{region " SIGNAL AREA : NAME->C_BMS_Wkup LENGTH->2 STARTBIT :44"}
_FB_CanTx_Message_Unpack_430.S_Bit_44		:= (GVL.IOVD.C_BMS_Wkup.x OR GVL.IOVD.C_BMS_Wkup.na) AND NOT GVL.IOVD.C_BMS_Wkup.e; 
_FB_CanTx_Message_Unpack_430.S_Bit_45		:= NOT GVL.IOVD.C_BMS_Wkup.v OR GVL.IOVD.C_BMS_Wkup.na OR GVL.IOVD.C_BMS_Wkup.e; 
{endregion}

{region " SIGNAL AREA : NAME->Z_Bat_Mode LENGTH->8 STARTBIT :48"}
_FB_CanTx_Message_Unpack_430.X_Byte_6					:=
(*SELECT 1 : Is data valid and range is not exceed?*)	SEL((GVL.IOVD.Z_Bat_Mode.v AND NOT GVL.IOVD.Z_Bat_Mode.RangeExcd),
(*SELECT 2 : Is NOT AVAILABLE ?*)						SEL(GVL.IOVD.Z_Bat_Mode.na,
(*SELECT 3 : Is ERROR active ?*)						SEL(GVL.IOVD.Z_Bat_Mode.e,
(*DEFAULT VALUE assignment*)							0,
(*ERROR is active*)										16#E),
(*NOT AVAILABLE is active*)								16#F),
(*Transmission is VALID*)								GVL.IOVD.Z_Bat_Mode.x);
{endregion}

{region " SIGNAL AREA : NAME->Z_ESS_Stat LENGTH->8 STARTBIT :56"}

_FB_CanTx_Message_Unpack_430.X_Byte_7					:=
(*SELECT 1 : Is data valid and range is not exceed?*)	SEL((GVL.IOVD.Z_ESS_Stat.v AND NOT GVL.IOVD.Z_ESS_Stat.RangeExcd),
(*SELECT 2 : Is NOT AVAILABLE ?*)						SEL(GVL.IOVD.Z_ESS_Stat.na,
(*SELECT 3 : Is ERROR active ?*)						SEL(GVL.IOVD.Z_ESS_Stat.e,
(*DEFAULT VALUE assignment*)							0,
(*ERROR is active*)										16#E),
(*NOT AVAILABLE is active*)								16#F),
(*Transmission is VALID*)								GVL.IOVD.Z_ESS_Stat.x);
{endregion}

_FB_CanTx_Message_Unpack_430.S_Bit_2 	:= TRUE;
_FB_CanTx_Message_Unpack_430.S_Bit_3 	:= TRUE;
_FB_CanTx_Message_Unpack_430.S_Bit_14 	:= TRUE;
_FB_CanTx_Message_Unpack_430.S_Bit_15 	:= TRUE;
_FB_CanTx_Message_Unpack_430.S_Bit_18	:= TRUE;
_FB_CanTx_Message_Unpack_430.S_Bit_19	:= TRUE;
_FB_CanTx_Message_Unpack_430.S_Bit_20	:= TRUE;
_FB_CanTx_Message_Unpack_430.S_Bit_21	:= TRUE;
_FB_CanTx_Message_Unpack_430.S_Bit_22	:= TRUE;
_FB_CanTx_Message_Unpack_430.S_Bit_23	:= TRUE;
_FB_CanTx_Message_Unpack_430.S_Bit_28	:= TRUE;
_FB_CanTx_Message_Unpack_430.S_Bit_29	:= TRUE;
_FB_CanTx_Message_Unpack_430.S_Bit_30	:= TRUE;
_FB_CanTx_Message_Unpack_430.S_Bit_31	:= TRUE;
_FB_CanTx_Message_Unpack_430.S_Bit_46	:= TRUE;
_FB_CanTx_Message_Unpack_430.S_Bit_47	:= TRUE;

_FB_CanTx_Message_Unpack_430 (		C_Enable		:= GVL.IOVD.C_En_ESS_Durum_0X430,
     								Obj_CAN			:= ADR(GVL.IC.Obj_CAN0),
     								X_MsgID			:= 16#430,
     								Tm_CycleTime	:= TIME#500MS,
     								N_Msg_Dlc		:= 8,
     								S_Extended		:= 0,
     								S_Sent_Ok   	=> GVL.IOVD.S_SentOk_ESS_Durum_0X430);
{endregion}
//-----------------------------------------------------------------------------------------------------------------------------
//-----------------------------------------------------------------------------------------------------------------------------
{region " MESSAGE AREA :ESS_Paket_Voltaji- ID:431"}

{region " SIGNAL AREA : NAME->X_U_Bat_1 LENGTH->16 STARTBIT :0"}
_FB_UNPACK_WORD_TO_BYTE_0 (
		X_WORD_0										:= 
(*SELECT 1 : Is data valid and range is not exceed?*)	SEL((GVL.IOVD.X_U_Bat_1.v AND NOT GVL.IOVD.X_U_Bat_1.RangeExcd),
(*SELECT 2 : Is NOT AVAILABLE ?*)						SEL(GVL.IOVD.X_U_Bat_1.na,
(*SELECT 3 : Is ERROR active ?*)						SEL(GVL.IOVD.X_U_Bat_1.e,
(*DEFAULT VALUE assignment*)							0,
(*ERROR is active*)										16#FEFE),
(*NOT AVAILABLE is active*)								16#FFFF),
(*Transmission is VALID*)								UINT_TO_WORD(REAL_TO_UINT((GVL.IOVD.X_U_Bat_1.x)/0.02))),
		X_BYTE_0										=> _FB_CanTx_Message_Unpack_431.X_Byte_0,
		X_BYTE_1										=> _FB_CanTx_Message_Unpack_431.X_Byte_1);
{endregion}

{region " SIGNAL AREA : NAME->X_U_Bat_2 LENGTH->16 STARTBIT :16"}
_FB_UNPACK_WORD_TO_BYTE_1 (
		X_WORD_0										:= 
(*SELECT 1 : Is data valid and range is not exceed?*)	SEL((GVL.IOVD.X_U_Bat_2.v AND NOT GVL.IOVD.X_U_Bat_2.RangeExcd),
(*SELECT 2 : Is NOT AVAILABLE ?*)						SEL(GVL.IOVD.X_U_Bat_2.na,
(*SELECT 3 : Is ERROR active ?*)						SEL(GVL.IOVD.X_U_Bat_2.e,
(*DEFAULT VALUE assignment*)							0,
(*ERROR is active*)										16#FEFE),
(*NOT AVAILABLE is active*)								16#FFFF),
(*Transmission is VALID*)								UINT_TO_WORD(REAL_TO_UINT((GVL.IOVD.X_U_Bat_2.x)/0.02))),
		X_BYTE_0										=> _FB_CanTx_Message_Unpack_431.X_Byte_2,
		X_BYTE_1										=> _FB_CanTx_Message_Unpack_431.X_Byte_3);
{endregion}

{region " SIGNAL AREA : NAME->X_U_Bat_3 LENGTH->16 STARTBIT :32"}
_FB_UNPACK_WORD_TO_BYTE_2 (
		X_WORD_0										:= 
(*SELECT 1 : Is data valid and range is not exceed?*)	SEL((GVL.IOVD.X_U_Bat_3.v AND NOT GVL.IOVD.X_U_Bat_3.RangeExcd),
(*SELECT 2 : Is NOT AVAILABLE ?*)						SEL(GVL.IOVD.X_U_Bat_3.na,
(*SELECT 3 : Is ERROR active ?*)						SEL(GVL.IOVD.X_U_Bat_3.e,
(*DEFAULT VALUE assignment*)							0,
(*ERROR is active*)										16#FEFE),
(*NOT AVAILABLE is active*)								16#FFFF),
(*Transmission is VALID*)								UINT_TO_WORD(REAL_TO_UINT((GVL.IOVD.X_U_Bat_3.x)/0.02))),
		X_BYTE_0										=> _FB_CanTx_Message_Unpack_431.X_Byte_4,
		X_BYTE_1										=> _FB_CanTx_Message_Unpack_431.X_Byte_5);
{endregion}

{region " SIGNAL AREA : NAME->X_U_Bat_4 LENGTH->16 STARTBIT :48"}
_FB_UNPACK_WORD_TO_BYTE_3 (
		X_WORD_0										:= 
(*SELECT 1 : Is data valid and range is not exceed?*)	SEL((GVL.IOVD.X_U_Bat_4.v AND NOT GVL.IOVD.X_U_Bat_4.RangeExcd),
(*SELECT 2 : Is NOT AVAILABLE ?*)						SEL(GVL.IOVD.X_U_Bat_4.na,
(*SELECT 3 : Is ERROR active ?*)						SEL(GVL.IOVD.X_U_Bat_4.e,
(*DEFAULT VALUE assignment*)							0,
(*ERROR is active*)										16#FEFE),
(*NOT AVAILABLE is active*)								16#FFFF),
(*Transmission is VALID*)								UINT_TO_WORD(REAL_TO_UINT((GVL.IOVD.X_U_Bat_4.x)/0.02))),
		X_BYTE_0										=> _FB_CanTx_Message_Unpack_431.X_Byte_6,
		X_BYTE_1										=> _FB_CanTx_Message_Unpack_431.X_Byte_7);
{endregion}

_FB_CanTx_Message_Unpack_431 (		C_Enable		:= GVL.IOVD.C_En_ESS_Paket_Voltaji_0X431,
     								Obj_CAN			:= ADR(GVL.IC.Obj_CAN0),
     								X_MsgID			:= 16#431,
     								Tm_CycleTime	:= TIME#500MS,
     								N_Msg_Dlc		:= 8,
     								S_Extended		:= 0,
     								S_Sent_Ok   	=> GVL.IOVD.S_SentOk_ESS_Paket_Voltaji_0X431);
{endregion}
//-----------------------------------------------------------------------------------------------------------------------------
//-----------------------------------------------------------------------------------------------------------------------------
{region " MESSAGE AREA :ESS_Paket_Akim- ID:432"}

{region " SIGNAL AREA : NAME->X_I_Bat_1 LENGTH->16 STARTBIT :0"}
_FB_UNPACK_WORD_TO_BYTE_4 (
		X_WORD_0										:= 
(*SELECT 1 : Is data valid and range is not exceed?*)	SEL((GVL.IOVD.X_I_Bat_1.v AND NOT GVL.IOVD.X_I_Bat_1.RangeExcd),
(*SELECT 2 : Is NOT AVAILABLE ?*)						SEL(GVL.IOVD.X_I_Bat_1.na,
(*SELECT 3 : Is ERROR active ?*)						SEL(GVL.IOVD.X_I_Bat_1.e,
(*DEFAULT VALUE assignment*)							UINT_TO_WORD(REAL_TO_UINT((3276.8)/0.1)),
(*ERROR is active*)										16#FEFE),
(*NOT AVAILABLE is active*)								16#FFFF),
(*Transmission is VALID*)								UINT_TO_WORD(REAL_TO_UINT((GVL.IOVD.X_I_Bat_1.x + 3276.8) / 0.1))),
		X_BYTE_0										=> _FB_CanTx_Message_432.X_Byte_0,
		X_BYTE_1										=> _FB_CanTx_Message_432.X_Byte_1);
{endregion}

{region " SIGNAL AREA : NAME->X_I_Bat_2 LENGTH->16 STARTBIT :16"}
_FB_UNPACK_WORD_TO_BYTE_5 (
		X_WORD_0										:= 
(*SELECT 1 : Is data valid and range is not exceed?*)	SEL((GVL.IOVD.X_I_Bat_2.v AND NOT GVL.IOVD.X_I_Bat_2.RangeExcd),
(*SELECT 2 : Is NOT AVAILABLE ?*)						SEL(GVL.IOVD.X_I_Bat_2.na,
(*SELECT 3 : Is ERROR active ?*)						SEL(GVL.IOVD.X_I_Bat_2.e,
(*DEFAULT VALUE assignment*)							UINT_TO_WORD(REAL_TO_UINT((3276.8)/0.1)),
(*ERROR is active*)										16#FEFE),
(*NOT AVAILABLE is active*)								16#FFFF),
(*Transmission is VALID*)								UINT_TO_WORD(REAL_TO_UINT((GVL.IOVD.X_I_Bat_2.x + 3276.8) / 0.1))),
		X_BYTE_0										=> _FB_CanTx_Message_432.X_Byte_2,
		X_BYTE_1										=> _FB_CanTx_Message_432.X_Byte_3);
{endregion}

{region " SIGNAL AREA : NAME->X_I_Bat_3 LENGTH->16 STARTBIT :32"}
_FB_UNPACK_WORD_TO_BYTE_6 (
		X_WORD_0										:= 
(*SELECT 1 : Is data valid and range is not exceed?*)	SEL((GVL.IOVD.X_I_Bat_3.v AND NOT GVL.IOVD.X_I_Bat_3.RangeExcd),
(*SELECT 2 : Is NOT AVAILABLE ?*)						SEL(GVL.IOVD.X_I_Bat_3.na,
(*SELECT 3 : Is ERROR active ?*)						SEL(GVL.IOVD.X_I_Bat_3.e,
(*DEFAULT VALUE assignment*)							UINT_TO_WORD(REAL_TO_UINT((3276.8)/0.1)),
(*ERROR is active*)										16#FEFE),
(*NOT AVAILABLE is active*)								16#FFFF),
(*Transmission is VALID*)								UINT_TO_WORD(REAL_TO_UINT((GVL.IOVD.X_I_Bat_3.x + 3276.8) / 0.1))),
		X_BYTE_0										=> _FB_CanTx_Message_432.X_Byte_4,
		X_BYTE_1										=> _FB_CanTx_Message_432.X_Byte_5);
{endregion}

{region " SIGNAL AREA : NAME->X_I_Bat_4 LENGTH->16 STARTBIT :48"}
_FB_UNPACK_WORD_TO_BYTE_7 (
		X_WORD_0										:= 
(*SELECT 1 : Is data valid and range is not exceed?*)	SEL((GVL.IOVD.X_I_Bat_4.v AND NOT GVL.IOVD.X_I_Bat_4.RangeExcd),
(*SELECT 2 : Is NOT AVAILABLE ?*)						SEL(GVL.IOVD.X_I_Bat_4.na,
(*SELECT 3 : Is ERROR active ?*)						SEL(GVL.IOVD.X_I_Bat_4.e,
(*DEFAULT VALUE assignment*)							UINT_TO_WORD(REAL_TO_UINT((3276.8)/0.1)),
(*ERROR is active*)										16#FEFE),
(*NOT AVAILABLE is active*)								16#FFFF),
(*Transmission is VALID*)								UINT_TO_WORD(REAL_TO_UINT((GVL.IOVD.X_I_Bat_4.x + 3276.8) / 0.1))),
		X_BYTE_0										=> _FB_CanTx_Message_432.X_Byte_6,
		X_BYTE_1										=> _FB_CanTx_Message_432.X_Byte_7);
{endregion}

_FB_CanTx_Message_432 (		C_Enable		:= GVL.IOVD.C_En_ESS_Paket_Akim_0X432,
     						Obj_CAN			:= ADR(GVL.IC.Obj_CAN0),
     						X_MsgID			:= 16#432,
     						Tm_CycleTime	:= TIME#500MS,
     						N_Msg_Dlc		:= 8,
     						S_Extended		:= 0,
     						S_Sent_Ok  	 	=> GVL.IOVD.S_SentOk_ESS_Paket_Akim_0X432);
{endregion}
//-----------------------------------------------------------------------------------------------------------------------------
//-----------------------------------------------------------------------------------------------------------------------------
{region " MESSAGE AREA :ESS_Maksimum_Hucre_Voltaji- ID:433"}

{region " SIGNAL AREA : NAME->X_U_Max_Cell_1 LENGTH->16 STARTBIT :0"}
_FB_UNPACK_WORD_TO_BYTE_8 (
		X_WORD_0										:= 
(*SELECT 1 : Is data valid and range is not exceed?*)	SEL((GVL.IOVD.X_U_Max_Bat_1.v AND NOT GVL.IOVD.X_U_Max_Bat_1.RangeExcd),
(*SELECT 2 : Is NOT AVAILABLE ?*)						SEL(GVL.IOVD.X_U_Max_Bat_1.na,
(*SELECT 3 : Is ERROR active ?*)						SEL(GVL.IOVD.X_U_Max_Bat_1.e,
(*DEFAULT VALUE assignment*)							0,
(*ERROR is active*)										16#FEFE),
(*NOT AVAILABLE is active*)								16#FFFF),
(*Transmission is VALID*)								UINT_TO_WORD(REAL_TO_UINT((GVL.IOVD.X_U_Max_Bat_1.x) / 0.1))),
		X_BYTE_0										=> _FB_CanTx_Message_433.X_Byte_0,
		X_BYTE_1										=> _FB_CanTx_Message_433.X_Byte_1);
{endregion}

{region " SIGNAL AREA : NAME->X_U_Max_Cell_2 LENGTH->16 STARTBIT :16"}
_FB_UNPACK_WORD_TO_BYTE_9 (
		X_WORD_0										:= 
(*SELECT 1 : Is data valid and range is not exceed?*)	SEL((GVL.IOVD.X_U_Max_Bat_2.v AND NOT GVL.IOVD.X_U_Max_Bat_2.RangeExcd),
(*SELECT 2 : Is NOT AVAILABLE ?*)						SEL(GVL.IOVD.X_U_Max_Bat_2.na,
(*SELECT 3 : Is ERROR active ?*)						SEL(GVL.IOVD.X_U_Max_Bat_2.e,
(*DEFAULT VALUE assignment*)							0,
(*ERROR is active*)										16#FEFE),
(*NOT AVAILABLE is active*)								16#FFFF),
(*Transmission is VALID*)								UINT_TO_WORD(REAL_TO_UINT((GVL.IOVD.X_U_Max_Bat_2.x) / 0.1))),
		X_BYTE_0										=> _FB_CanTx_Message_433.X_Byte_2,
		X_BYTE_1										=> _FB_CanTx_Message_433.X_Byte_3);
{endregion}

{region " SIGNAL AREA : NAME->X_U_Max_Cell_3 LENGTH->16 STARTBIT :32"}
_FB_UNPACK_WORD_TO_BYTE_10 (
		X_WORD_0										:= 
(*SELECT 1 : Is data valid and range is not exceed?*)	SEL((GVL.IOVD.X_U_Max_Bat_3.v AND NOT GVL.IOVD.X_U_Max_Bat_3.RangeExcd),
(*SELECT 2 : Is NOT AVAILABLE ?*)						SEL(GVL.IOVD.X_U_Max_Bat_3.na,
(*SELECT 3 : Is ERROR active ?*)						SEL(GVL.IOVD.X_U_Max_Bat_3.e,
(*DEFAULT VALUE assignment*)							0,
(*ERROR is active*)										16#FEFE),
(*NOT AVAILABLE is active*)								16#FFFF),
(*Transmission is VALID*)								UINT_TO_WORD(REAL_TO_UINT((GVL.IOVD.X_U_Max_Bat_3.x) / 0.1))),
		X_BYTE_0										=> _FB_CanTx_Message_433.X_Byte_4,
		X_BYTE_1										=> _FB_CanTx_Message_433.X_Byte_5);
{endregion}

{region " SIGNAL AREA : NAME->X_U_Max_Cell_4 LENGTH->16 STARTBIT :48"}
_FB_UNPACK_WORD_TO_BYTE_11 (
		X_WORD_0										:= 
(*SELECT 1 : Is data valid and range is not exceed?*)	SEL((GVL.IOVD.X_U_Max_Bat_4.v AND NOT GVL.IOVD.X_U_Max_Bat_4.RangeExcd),
(*SELECT 2 : Is NOT AVAILABLE ?*)						SEL(GVL.IOVD.X_U_Max_Bat_4.na,
(*SELECT 3 : Is ERROR active ?*)						SEL(GVL.IOVD.X_U_Max_Bat_4.e,
(*DEFAULT VALUE assignment*)							0,
(*ERROR is active*)										16#FEFE),
(*NOT AVAILABLE is active*)								16#FFFF),
(*Transmission is VALID*)								UINT_TO_WORD(REAL_TO_UINT((GVL.IOVD.X_U_Max_Bat_4.x) / 0.1))),
		X_BYTE_0										=> _FB_CanTx_Message_433.X_Byte_6,
		X_BYTE_1										=> _FB_CanTx_Message_433.X_Byte_7);
{endregion}

_FB_CanTx_Message_433 (		C_Enable		:= GVL.IOVD.C_En_ESS_Maksimum_Hucre_Voltaji_0X433,
     						Obj_CAN			:= ADR(GVL.IC.Obj_CAN0),
     						X_MsgID			:= 16#433,
     						Tm_CycleTime	:= TIME#500MS,
     						N_Msg_Dlc		:= 8,
     						S_Extended		:= 0,
     						S_Sent_Ok   	=> GVL.IOVD.S_SentOk_ESS_Maksimum_Hucre_Voltaji_0X433);
{endregion}
//-----------------------------------------------------------------------------------------------------------------------------
//-----------------------------------------------------------------------------------------------------------------------------
{region " MESSAGE AREA :ESS_Minimum_Hucre_Voltaji- ID:434"}

{region " SIGNAL AREA : NAME->X_U_Min_Cell_1 LENGTH->16 STARTBIT :0"}
_FB_UNPACK_WORD_TO_BYTE_12 (
		X_WORD_0										:= 
(*SELECT 1 : Is data valid and range is not exceed?*)	SEL((GVL.IOVD.X_U_Min_Bat_1.v AND NOT GVL.IOVD.X_U_Min_Bat_1.RangeExcd),
(*SELECT 2 : Is NOT AVAILABLE ?*)						SEL(GVL.IOVD.X_U_Min_Bat_1.na,
(*SELECT 3 : Is ERROR active ?*)						SEL(GVL.IOVD.X_U_Min_Bat_1.e,
(*DEFAULT VALUE assignment*)							0,
(*ERROR is active*)										16#FEFE),
(*NOT AVAILABLE is active*)								16#FFFF),
(*Transmission is VALID*)								UINT_TO_WORD(REAL_TO_UINT((GVL.IOVD.X_U_Min_Bat_1.x) / 0.1))),
		X_BYTE_0										=> _FB_CanTx_Message_Unpack_434.X_Byte_0,
		X_BYTE_1										=> _FB_CanTx_Message_Unpack_434.X_Byte_1);
{endregion}

{region " SIGNAL AREA : NAME->X_U_Min_Cell_2 LENGTH->16 STARTBIT :16"}
_FB_UNPACK_WORD_TO_BYTE_13 (
		X_WORD_0										:= 
(*SELECT 1 : Is data valid and range is not exceed?*)	SEL((GVL.IOVD.X_U_Min_Bat_2.v AND NOT GVL.IOVD.X_U_Min_Bat_2.RangeExcd),
(*SELECT 2 : Is NOT AVAILABLE ?*)						SEL(GVL.IOVD.X_U_Min_Bat_2.na,
(*SELECT 3 : Is ERROR active ?*)						SEL(GVL.IOVD.X_U_Min_Bat_2.e,
(*DEFAULT VALUE assignment*)							0,
(*ERROR is active*)										16#FEFE),
(*NOT AVAILABLE is active*)								16#FFFF),
(*Transmission is VALID*)								UINT_TO_WORD(REAL_TO_UINT((GVL.IOVD.X_U_Min_Bat_2.x) / 0.1))),
		X_BYTE_0										=> _FB_CanTx_Message_Unpack_434.X_Byte_2,
		X_BYTE_1										=> _FB_CanTx_Message_Unpack_434.X_Byte_3);
{endregion}

{region " SIGNAL AREA : NAME->X_U_Min_Cell_3 LENGTH->16 STARTBIT :32"}
_FB_UNPACK_WORD_TO_BYTE_14 (
		X_WORD_0										:= 
(*SELECT 1 : Is data valid and range is not exceed?*)	SEL((GVL.IOVD.X_U_Min_Bat_3.v AND NOT GVL.IOVD.X_U_Min_Bat_3.RangeExcd),
(*SELECT 2 : Is NOT AVAILABLE ?*)						SEL(GVL.IOVD.X_U_Min_Bat_3.na,
(*SELECT 3 : Is ERROR active ?*)						SEL(GVL.IOVD.X_U_Min_Bat_3.e,
(*DEFAULT VALUE assignment*)							0,
(*ERROR is active*)										16#FEFE),
(*NOT AVAILABLE is active*)								16#FFFF),
(*Transmission is VALID*)								UINT_TO_WORD(REAL_TO_UINT((GVL.IOVD.X_U_Min_Bat_3.x) / 0.1))),
		X_BYTE_0										=> _FB_CanTx_Message_Unpack_434.X_Byte_4,
		X_BYTE_1										=> _FB_CanTx_Message_Unpack_434.X_Byte_5);
{endregion}

{region " SIGNAL AREA : NAME->X_U_Min_Cell_4 LENGTH->16 STARTBIT :48"}
_FB_UNPACK_WORD_TO_BYTE_15 (
		X_WORD_0										:= 
(*SELECT 1 : Is data valid and range is not exceed?*)	SEL((GVL.IOVD.X_U_Min_Bat_4.v AND NOT GVL.IOVD.X_U_Min_Bat_4.RangeExcd),
(*SELECT 2 : Is NOT AVAILABLE ?*)						SEL(GVL.IOVD.X_U_Min_Bat_4.na,
(*SELECT 3 : Is ERROR active ?*)						SEL(GVL.IOVD.X_U_Min_Bat_4.e,
(*DEFAULT VALUE assignment*)							0,
(*ERROR is active*)										16#FEFE),
(*NOT AVAILABLE is active*)								16#FFFF),
(*Transmission is VALID*)								UINT_TO_WORD(REAL_TO_UINT((GVL.IOVD.X_U_Min_Bat_4.x) / 0.1))),
		X_BYTE_0										=> _FB_CanTx_Message_Unpack_434.X_Byte_6,
		X_BYTE_1										=> _FB_CanTx_Message_Unpack_434.X_Byte_7);
{endregion}

_FB_CanTx_Message_Unpack_434 (		C_Enable		:= GVL.IOVD.C_En_ESS_Minimum_Hucre_Voltaji_0X434,
     								Obj_CAN			:= ADR(GVL.IC.Obj_CAN0),
     								X_MsgID			:= 16#434,
     								Tm_CycleTime	:= TIME#500MS,
     								N_Msg_Dlc		:= 8,
     								S_Extended		:= 0,
     								S_Sent_Ok   	=> GVL.IOVD.S_SentOk_ESS_Minimum_Hucre_Voltaji_0X434);
{endregion}
//-----------------------------------------------------------------------------------------------------------------------------
//-----------------------------------------------------------------------------------------------------------------------------
{region " MESSAGE AREA :ESS_Ortalama_Hucre_Voltaji- ID:435"}

{region " SIGNAL AREA : NAME->X_U_Avg_Cell_1 LENGTH->16 STARTBIT :0"}
_FB_UNPACK_WORD_TO_BYTE_16 (
		X_WORD_0										:= 
(*SELECT 1 : Is data valid and range is not exceed?*)	SEL((GVL.IOVD.X_U_Avg_Cell_1.v AND NOT GVL.IOVD.X_U_Avg_Cell_1.RangeExcd),
(*SELECT 2 : Is NOT AVAILABLE ?*)						SEL(GVL.IOVD.X_U_Avg_Cell_1.na,
(*SELECT 3 : Is ERROR active ?*)						SEL(GVL.IOVD.X_U_Avg_Cell_1.e,
(*DEFAULT VALUE assignment*)							0,
(*ERROR is active*)										16#FEFE),
(*NOT AVAILABLE is active*)								16#FFFF),
(*Transmission is VALID*)								UINT_TO_WORD(REAL_TO_UINT((GVL.IOVD.X_U_Avg_Cell_1.x)/0.01))),
		X_BYTE_0										=> _FB_CanTx_Message_435.X_Byte_0,
		X_BYTE_1										=> _FB_CanTx_Message_435.X_Byte_1);
{endregion}

{region " SIGNAL AREA : NAME->X_U_Avg_Cell_2 LENGTH->16 STARTBIT :16"}
_FB_UNPACK_WORD_TO_BYTE_17 (
		X_WORD_0										:= 
(*SELECT 1 : Is data valid and range is not exceed?*)	SEL((GVL.IOVD.X_U_Avg_Cell_2.v AND NOT GVL.IOVD.X_U_Avg_Cell_2.RangeExcd),
(*SELECT 2 : Is NOT AVAILABLE ?*)						SEL(GVL.IOVD.X_U_Avg_Cell_2.na,
(*SELECT 3 : Is ERROR active ?*)						SEL(GVL.IOVD.X_U_Avg_Cell_2.e,
(*DEFAULT VALUE assignment*)							0,
(*ERROR is active*)										16#FEFE),
(*NOT AVAILABLE is active*)								16#FFFF),
(*Transmission is VALID*)								UINT_TO_WORD(REAL_TO_UINT((GVL.IOVD.X_U_Avg_Cell_2.x)/0.01))),
		X_BYTE_0										=> _FB_CanTx_Message_435.X_Byte_2,
		X_BYTE_1										=> _FB_CanTx_Message_435.X_Byte_3);
{endregion}

{region " SIGNAL AREA : NAME->X_U_Avg_Cell_3 LENGTH->16 STARTBIT :32"}
_FB_UNPACK_WORD_TO_BYTE_18 (
		X_WORD_0										:= 
(*SELECT 1 : Is data valid and range is not exceed?*)	SEL((GVL.IOVD.X_U_Avg_Cell_3.v AND NOT GVL.IOVD.X_U_Avg_Cell_3.RangeExcd),
(*SELECT 2 : Is NOT AVAILABLE ?*)						SEL(GVL.IOVD.X_U_Avg_Cell_3.na,
(*SELECT 3 : Is ERROR active ?*)						SEL(GVL.IOVD.X_U_Avg_Cell_3.e,
(*DEFAULT VALUE assignment*)							0,
(*ERROR is active*)										16#FEFE),
(*NOT AVAILABLE is active*)								16#FFFF),
(*Transmission is VALID*)								UINT_TO_WORD(REAL_TO_UINT((GVL.IOVD.X_U_Avg_Cell_3.x)/0.01))),
		X_BYTE_0										=> _FB_CanTx_Message_435.X_Byte_4,
		X_BYTE_1										=> _FB_CanTx_Message_435.X_Byte_5);
{endregion}

{region " SIGNAL AREA : NAME->X_U_Avg_Cell_4 LENGTH->16 STARTBIT :48"}
_FB_UNPACK_WORD_TO_BYTE_19 (
		X_WORD_0										:= 
(*SELECT 1 : Is data valid and range is not exceed?*)	SEL((GVL.IOVD.X_U_Avg_Cell_4.v AND NOT GVL.IOVD.X_U_Avg_Cell_4.RangeExcd),
(*SELECT 2 : Is NOT AVAILABLE ?*)						SEL(GVL.IOVD.X_U_Avg_Cell_4.na,
(*SELECT 3 : Is ERROR active ?*)						SEL(GVL.IOVD.X_U_Avg_Cell_4.e,
(*DEFAULT VALUE assignment*)							0,
(*ERROR is active*)										16#FEFE),
(*NOT AVAILABLE is active*)								16#FFFF),
(*Transmission is VALID*)								UINT_TO_WORD(REAL_TO_UINT((GVL.IOVD.X_U_Avg_Cell_4.x)/0.01))),
		X_BYTE_0										=> _FB_CanTx_Message_435.X_Byte_6,
		X_BYTE_1										=> _FB_CanTx_Message_435.X_Byte_7);
{endregion}

_FB_CanTx_Message_435 (		C_Enable		:= GVL.IOVD.C_En_ESS_Ortalama_Hucre_Voltaji_0X435,
     						Obj_CAN			:= ADR(GVL.IC.Obj_CAN0),
     						X_MsgID			:= 16#435,
     						Tm_CycleTime	:= TIME#500MS,
     						N_Msg_Dlc		:= 8,
     						S_Extended		:= 0,
     						S_Sent_Ok   	=> GVL.IOVD.S_SentOk_ESS_Ortalama_Hucre_Voltaji_0X435);
{endregion}
//-----------------------------------------------------------------------------------------------------------------------------
//-----------------------------------------------------------------------------------------------------------------------------
{region " MESSAGE AREA :ESS_Sicaklik- ID:436"}

{region " SIGNAL AREA : NAME->X_T_Max_Cell_1 LENGTH->8 STARTBIT :0"}
_FB_CanTx_Message_436.X_Byte_0							:=
(*SELECT 1 : Is data valid and range is not exceed?*)	SEL((GVL.IOVD.X_T_Max_Bat_1.v AND NOT GVL.IOVD.X_T_Max_Bat_1.RangeExcd),
(*SELECT 2 : Is NOT AVAILABLE ?*)						SEL(GVL.IOVD.X_T_Max_Bat_1.na,
(*SELECT 3 : Is ERROR active ?*)						SEL(GVL.IOVD.X_T_Max_Bat_1.e,
(*DEFAULT VALUE assignment*)							USINT_TO_BYTE(REAL_TO_USINT((40))),
(*ERROR is active*)										16#FE),
(*NOT AVAILABLE is active*)								16#FF),
(*Transmission is VALID*)								USINT_TO_BYTE(REAL_TO_USINT((GVL.IOVD.X_T_Max_Bat_1.x + 40))));
{endregion}

{region " SIGNAL AREA : NAME->X_T_Max_Cell_2 LENGTH->8 STARTBIT :8"}
_FB_CanTx_Message_436.X_Byte_1							:=
(*SELECT 1 : Is data valid and range is not exceed?*)	SEL((GVL.IOVD.X_T_Max_Bat_2.v AND NOT GVL.IOVD.X_T_Max_Bat_2.RangeExcd),
(*SELECT 2 : Is NOT AVAILABLE ?*)						SEL(GVL.IOVD.X_T_Max_Bat_2.na,
(*SELECT 3 : Is ERROR active ?*)						SEL(GVL.IOVD.X_T_Max_Bat_2.e,
(*DEFAULT VALUE assignment*)							USINT_TO_BYTE(REAL_TO_USINT((40))),
(*ERROR is active*)										16#FE),
(*NOT AVAILABLE is active*)								16#FF),
(*Transmission is VALID*)								USINT_TO_BYTE(REAL_TO_USINT((GVL.IOVD.X_T_Max_Bat_2.x + 40))));
{endregion}

{region " SIGNAL AREA : NAME->X_T_Max_Cell_3 LENGTH->8 STARTBIT :16"}
_FB_CanTx_Message_436.X_Byte_2							:=
(*SELECT 1 : Is data valid and range is not exceed?*)	SEL((GVL.IOVD.X_T_Max_Bat_3.v AND NOT GVL.IOVD.X_T_Max_Bat_3.RangeExcd),
(*SELECT 2 : Is NOT AVAILABLE ?*)						SEL(GVL.IOVD.X_T_Max_Bat_3.na,
(*SELECT 3 : Is ERROR active ?*)						SEL(GVL.IOVD.X_T_Max_Bat_3.e,
(*DEFAULT VALUE assignment*)							USINT_TO_BYTE(REAL_TO_USINT((40))),
(*ERROR is active*)										16#FE),
(*NOT AVAILABLE is active*)								16#FF),
(*Transmission is VALID*)								USINT_TO_BYTE(REAL_TO_USINT((GVL.IOVD.X_T_Max_Bat_3.x + 40))));
{endregion}

{region " SIGNAL AREA : NAME->X_T_Min_Cell_1 LENGTH->8 STARTBIT :32"}
_FB_CanTx_Message_436.X_Byte_4							:=
(*SELECT 1 : Is data valid and range is not exceed?*)	SEL((GVL.IOVD.X_T_Min_Bat_1.v AND NOT GVL.IOVD.X_T_Min_Bat_1.RangeExcd),
(*SELECT 2 : Is NOT AVAILABLE ?*)						SEL(GVL.IOVD.X_T_Min_Bat_1.na,
(*SELECT 3 : Is ERROR active ?*)						SEL(GVL.IOVD.X_T_Min_Bat_1.e,
(*DEFAULT VALUE assignment*)							USINT_TO_BYTE(REAL_TO_USINT((40))),
(*ERROR is active*)										16#FE),
(*NOT AVAILABLE is active*)								16#FF),
(*Transmission is VALID*)								USINT_TO_BYTE(REAL_TO_USINT((GVL.IOVD.X_T_Min_Bat_1.x + 40))));
{endregion}

{region " SIGNAL AREA : NAME->X_T_Min_Cell_2 LENGTH->8 STARTBIT :40"}
_FB_CanTx_Message_436.X_Byte_5							:=
(*SELECT 1 : Is data valid and range is not exceed?*)	SEL((GVL.IOVD.X_T_Min_Bat_2.v AND NOT GVL.IOVD.X_T_Min_Bat_2.RangeExcd),
(*SELECT 2 : Is NOT AVAILABLE ?*)						SEL(GVL.IOVD.X_T_Min_Bat_2.na,
(*SELECT 3 : Is ERROR active ?*)						SEL(GVL.IOVD.X_T_Min_Bat_2.e,
(*DEFAULT VALUE assignment*)							USINT_TO_BYTE(REAL_TO_USINT((40))),
(*ERROR is active*)										16#FE),
(*NOT AVAILABLE is active*)								16#FF),
(*Transmission is VALID*)								USINT_TO_BYTE(REAL_TO_USINT((GVL.IOVD.X_T_Min_Bat_2.x + 40))));
{endregion}

{region " SIGNAL AREA : NAME->X_T_Min_Cell_3 LENGTH->8 STARTBIT :48"}
_FB_CanTx_Message_436.X_Byte_6							:=
(*SELECT 1 : Is data valid and range is not exceed?*)	SEL((GVL.IOVD.X_T_Min_Bat_3.v AND NOT GVL.IOVD.X_T_Min_Bat_3.RangeExcd),
(*SELECT 2 : Is NOT AVAILABLE ?*)						SEL(GVL.IOVD.X_T_Min_Bat_3.na,
(*SELECT 3 : Is ERROR active ?*)						SEL(GVL.IOVD.X_T_Min_Bat_3.e,
(*DEFAULT VALUE assignment*)							USINT_TO_BYTE(REAL_TO_USINT((40))),
(*ERROR is active*)										16#FE),
(*NOT AVAILABLE is active*)								16#FF),
(*Transmission is VALID*)								USINT_TO_BYTE(REAL_TO_USINT((GVL.IOVD.X_T_Min_Bat_3.x + 40))));
{endregion}

{region " SIGNAL AREA : NAME->X_T_Min_Cell_4 LENGTH->8 STARTBIT :56"}
_FB_CanTx_Message_436.X_Byte_7							:=
(*SELECT 1 : Is data valid and range is not exceed?*)	SEL((GVL.IOVD.X_T_Avg_Bat_1.v AND NOT GVL.IOVD.X_T_Avg_Bat_1.RangeExcd),
(*SELECT 2 : Is NOT AVAILABLE ?*)						SEL(GVL.IOVD.X_T_Avg_Bat_1.na,
(*SELECT 3 : Is ERROR active ?*)						SEL(GVL.IOVD.X_T_Avg_Bat_1.e,
(*DEFAULT VALUE assignment*)							USINT_TO_BYTE(REAL_TO_USINT((40))),
(*ERROR is active*)										16#FE),
(*NOT AVAILABLE is active*)								16#FF),
(*Transmission is VALID*)								USINT_TO_BYTE(REAL_TO_USINT((GVL.IOVD.X_T_Avg_Bat_1.x + 40))));
{endregion}

_FB_CanTx_Message_436.X_Byte_3				:= 16#FF;

_FB_CanTx_Message_436 (		C_Enable		:= GVL.IOVD.C_En_ESS_Sicaklik_0X436,
     						Obj_CAN			:= ADR(GVL.IC.Obj_CAN0),
     						X_MsgID			:= 16#436,
     						Tm_CycleTime	:= TIME#500MS,
     						N_Msg_Dlc		:= 8,
     						S_Extended		:= 0,
     						S_Sent_Ok  	 	=> GVL.IOVD.S_SentOk_ESS_Sicaklik_0X436);
{endregion}
//-----------------------------------------------------------------------------------------------------------------------------
//-----------------------------------------------------------------------------------------------------------------------------
{region " MESSAGE AREA :ESS_Analog- ID:437"}

{region " SIGNAL AREA : NAME->X_I_Max_Chrg LENGTH->16 STARTBIT :16"}
_FB_UNPACK_WORD_TO_BYTE_20 (
		X_WORD_0										:= 
(*SELECT 1 : Is data valid and range is not exceed?*)	SEL((GVL.IOVD.X_I_Max_Chrg.v AND NOT GVL.IOVD.X_I_Max_Chrg.RangeExcd),
(*SELECT 2 : Is NOT AVAILABLE ?*)						SEL(GVL.IOVD.X_I_Max_Chrg.na,
(*SELECT 3 : Is ERROR active ?*)						SEL(GVL.IOVD.X_I_Max_Chrg.e,
(*DEFAULT VALUE assignment*)							UINT_TO_WORD(REAL_TO_UINT((3000)/0.1)),
(*ERROR is active*)										16#FEFE),
(*NOT AVAILABLE is active*)								16#FFFF),
(*Transmission is VALID*)								UINT_TO_WORD(REAL_TO_UINT((GVL.IOVD.X_I_Max_Chrg.x + 3000)/0.1))),
		X_BYTE_0										=> _FB_CanTx_Message_Unpack_437.X_Byte_2,
		X_BYTE_1										=> _FB_CanTx_Message_Unpack_437.X_Byte_3);
{endregion}

{region " SIGNAL AREA : NAME->X_I_Max_Dischrg LENGTH->16 STARTBIT :32"}
_FB_UNPACK_WORD_TO_BYTE_21 (
		X_WORD_0										:= 
(*SELECT 1 : Is data valid and range is not exceed?*)	SEL((GVL.IOVD.X_I_Max_Dischrg.v AND NOT GVL.IOVD.X_I_Max_Dischrg.RangeExcd),
(*SELECT 2 : Is NOT AVAILABLE ?*)						SEL(GVL.IOVD.X_I_Max_Dischrg.na,
(*SELECT 3 : Is ERROR active ?*)						SEL(GVL.IOVD.X_I_Max_Dischrg.e,
(*DEFAULT VALUE assignment*)							UINT_TO_WORD(REAL_TO_UINT((3000)/0.1)),
(*ERROR is active*)										16#FEFE),
(*NOT AVAILABLE is active*)								16#FFFF),
(*Transmission is VALID*)								UINT_TO_WORD(REAL_TO_UINT((GVL.IOVD.X_I_Max_Dischrg.x + 3000)/0.1))),
		X_BYTE_0										=> _FB_CanTx_Message_Unpack_437.X_Byte_4,
		X_BYTE_1										=> _FB_CanTx_Message_Unpack_437.X_Byte_5);
{endregion}

{region " SIGNAL AREA : NAME->X_U_Tot_Bat LENGTH->16 STARTBIT :48"}
_FB_UNPACK_WORD_TO_BYTE_22 (
		X_WORD_0										:= 
(*SELECT 1 : Is data valid and range is not exceed?*)	SEL((GVL.IOVD.X_U_Tot_Bat.v AND NOT GVL.IOVD.X_U_Tot_Bat.RangeExcd),
(*SELECT 2 : Is NOT AVAILABLE ?*)						SEL(GVL.IOVD.X_U_Tot_Bat.na,
(*SELECT 3 : Is ERROR active ?*)						SEL(GVL.IOVD.X_U_Tot_Bat.e,
(*DEFAULT VALUE assignment*)							0,
(*ERROR is active*)										16#FEFE),
(*NOT AVAILABLE is active*)								16#FFFF),
(*Transmission is VALID*)								UINT_TO_WORD(REAL_TO_UINT((GVL.IOVD.X_U_Tot_Bat.x)/0.1))),
		X_BYTE_0										=> _FB_CanTx_Message_Unpack_437.X_Byte_6,
		X_BYTE_1										=> _FB_CanTx_Message_Unpack_437.X_Byte_7);
{endregion}

_FB_CanTx_Message_Unpack_437.X_Byte_0			:= 16#FF;
_FB_CanTx_Message_Unpack_437.X_Byte_1			:= 16#FF;

_FB_CanTx_Message_Unpack_437 (		C_Enable		:= GVL.IOVD.C_En_ESS_Analog_0X437,
     								Obj_CAN			:= ADR(GVL.IC.Obj_CAN0),
     								X_MsgID			:= 16#437,
     								Tm_CycleTime	:= TIME#500MS,
     								N_Msg_Dlc		:= 8,
     								S_Extended		:= 0,
     								S_Sent_Ok   	=> GVL.IOVD.S_SentOk_ESS_Analog_0X437);
{endregion}
//-----------------------------------------------------------------------------------------------------------------------------
//-----------------------------------------------------------------------------------------------------------------------------
{region " MESSAGE AREA :ESS_Sogutma_Suyu- ID:438"}

{region " SIGNAL AREA : NAME->W_T_Clt LENGTH->8 STARTBIT :0"}
_FB_CanTx_Message_438.X_Byte_0							:=
(*SELECT 1 : Is data valid and range is not exceed?*)	SEL((GVL.IOVD.W_T_Clt.v AND NOT GVL.IOVD.W_T_Clt.RangeExcd),
(*SELECT 2 : Is NOT AVAILABLE ?*)						SEL(GVL.IOVD.W_T_Clt.na,
(*SELECT 3 : Is ERROR active ?*)						SEL(GVL.IOVD.W_T_Clt.e,
(*DEFAULT VALUE assignment*)							USINT_TO_BYTE(REAL_TO_USINT((40))),
(*ERROR is active*)										16#FE),
(*NOT AVAILABLE is active*)								16#FF),
(*Transmission is VALID*)								USINT_TO_BYTE(REAL_TO_USINT((GVL.IOVD.W_T_Clt.x + 40))));
{endregion}

{region " SIGNAL AREA : NAME->X_T_Clt LENGTH->8 STARTBIT :8"}
_FB_CanTx_Message_438.X_Byte_1							:=
(*SELECT 1 : Is data valid and range is not exceed?*)	SEL((GVL.IOVD.X_T_Clt.v AND NOT GVL.IOVD.X_T_Clt.RangeExcd),
(*SELECT 2 : Is NOT AVAILABLE ?*)						SEL(GVL.IOVD.X_T_Clt.na,
(*SELECT 3 : Is ERROR active ?*)						SEL(GVL.IOVD.X_T_Clt.e,
(*DEFAULT VALUE assignment*)							USINT_TO_BYTE(REAL_TO_USINT((40))),
(*ERROR is active*)										16#FE),
(*NOT AVAILABLE is active*)								16#FF),
(*Transmission is VALID*)								USINT_TO_BYTE(REAL_TO_USINT((GVL.IOVD.X_T_Clt.x + 40))));
{endregion}

_FB_CanTx_Message_438.X_Byte_2 		:= 16#FF;
_FB_CanTx_Message_438.X_Byte_3		:= 16#FF;
_FB_CanTx_Message_438.X_Byte_4		:= 16#FF;
_FB_CanTx_Message_438.X_Byte_5		:= 16#FF;
_FB_CanTx_Message_438.X_Byte_6		:= 16#FF;
_FB_CanTx_Message_438.X_Byte_7		:= 16#FF;
	 
_FB_CanTx_Message_438 (		C_Enable		:= GVL.IOVD.C_En_ESS_Sogutma_Suyu_0X438,
     						Obj_CAN			:= ADR(GVL.IC.Obj_CAN0),
     						X_MsgID			:= 16#438,
     						Tm_CycleTime	:= TIME#500MS,
     						N_Msg_Dlc		:= 8,
     						S_Extended		:= 0,
     						S_Sent_Ok   	=> GVL.IOVD.S_SentOk_ESS_Sogutma_Suyu_0X438);
{endregion}
//-----------------------------------------------------------------------------------------------------------------------------
//-----------------------------------------------------------------------------------------------------------------------------
{region " MESSAGE AREA :Sarj_Durum- ID:4A0"}

{region " SIGNAL AREA : NAME->S_Vh_Chrg_Perm LENGTH->2 STARTBIT :0"}
_FB_CanTx_Message_Unpack_4A0.S_Bit_0		:= (GVL.IOVD.S_Vh_Chrg_Perm.x OR GVL.IOVD.S_Vh_Chrg_Perm.na) AND NOT GVL.IOVD.S_Vh_Chrg_Perm.e; 
_FB_CanTx_Message_Unpack_4A0.S_Bit_1		:= NOT GVL.IOVD.S_Vh_Chrg_Perm.v OR GVL.IOVD.S_Vh_Chrg_Perm.na OR GVL.IOVD.S_Vh_Chrg_Perm.e; 
{endregion}

{region " SIGNAL AREA : NAME->S_Vh_Insu_Meas LENGTH->2 STARTBIT :2"}
_FB_CanTx_Message_Unpack_4A0.S_Bit_2		:= (GVL.IOVD.S_Vh_Insu_Meas.x OR GVL.IOVD.S_Vh_Insu_Meas.na) AND NOT GVL.IOVD.S_Vh_Insu_Meas.e; 
_FB_CanTx_Message_Unpack_4A0.S_Bit_3		:= NOT GVL.IOVD.S_Vh_Insu_Meas.v OR GVL.IOVD.S_Vh_Insu_Meas.na OR GVL.IOVD.S_Vh_Insu_Meas.e; 
{endregion}

{region " SIGNAL AREA : NAME->S_Vh_Mobil LENGTH->2 STARTBIT :4"}
_FB_CanTx_Message_Unpack_4A0.S_Bit_4		:= (GVL.IOVD.S_Vh_Mobil.x OR GVL.IOVD.S_Vh_Mobil.na) AND NOT GVL.IOVD.S_Vh_Mobil.e; 
_FB_CanTx_Message_Unpack_4A0.S_Bit_5		:= NOT GVL.IOVD.S_Vh_Mobil.v OR GVL.IOVD.S_Vh_Mobil.na OR GVL.IOVD.S_Vh_Mobil.e; 
{endregion}		   

{region " SIGNAL AREA : NAME->S_Chrg_Cmpl LENGTH->2 STARTBIT :8"}
_FB_CanTx_Message_Unpack_4A0.S_Bit_8		:= (GVL.IOVD.S_Chrg_Cmpl.x OR GVL.IOVD.S_Chrg_Cmpl.na) AND NOT GVL.IOVD.S_Chrg_Cmpl.e; 
_FB_CanTx_Message_Unpack_4A0.S_Bit_9		:= NOT GVL.IOVD.S_Chrg_Cmpl.v OR GVL.IOVD.S_Chrg_Cmpl.na OR GVL.IOVD.S_Chrg_Cmpl.e; 
{endregion}

{region " SIGNAL AREA : NAME->S_EV_Rdy LENGTH->2 STARTBIT :10"}
_FB_CanTx_Message_Unpack_4A0.S_Bit_10		:= (GVL.IOVD.S_EV_Rdy.x OR GVL.IOVD.S_EV_Rdy.na) AND NOT GVL.IOVD.S_EV_Rdy.e; 
_FB_CanTx_Message_Unpack_4A0.S_Bit_11		:= NOT GVL.IOVD.S_EV_Rdy.v OR GVL.IOVD.S_EV_Rdy.na OR GVL.IOVD.S_EV_Rdy.e; 
{endregion}

{region " SIGNAL AREA : NAME->C_Chrg_Btn_Lft_Bwd_Led_Ctrl LENGTH->2 STARTBIT :12"}
_FB_CanTx_Message_Unpack_4A0.S_Bit_12		:= (GVL.IOVD.C_Chrg_Btn_Lft_Bwd_Led_Ctrl.x OR GVL.IOVD.C_Chrg_Btn_Lft_Bwd_Led_Ctrl.na) AND NOT GVL.IOVD.C_Chrg_Btn_Lft_Bwd_Led_Ctrl.e; 
_FB_CanTx_Message_Unpack_4A0.S_Bit_13		:= NOT GVL.IOVD.C_Chrg_Btn_Lft_Bwd_Led_Ctrl.v OR GVL.IOVD.C_Chrg_Btn_Lft_Bwd_Led_Ctrl.na OR GVL.IOVD.C_Chrg_Btn_Lft_Bwd_Led_Ctrl.e; 
{endregion}

{region " SIGNAL AREA : NAME->S_Pnt_Chrg_Mode_Sel LENGTH->2 STARTBIT :16"}
_FB_CanTx_Message_Unpack_4A0.S_Bit_16		:= (GVL.IOVD.S_Pnt_Chrg_Mode_Sel.x OR GVL.IOVD.S_Pnt_Chrg_Mode_Sel.na) AND NOT GVL.IOVD.S_Pnt_Chrg_Mode_Sel.e; 
_FB_CanTx_Message_Unpack_4A0.S_Bit_17		:= NOT GVL.IOVD.S_Pnt_Chrg_Mode_Sel.v OR GVL.IOVD.S_Pnt_Chrg_Mode_Sel.na OR GVL.IOVD.S_Pnt_Chrg_Mode_Sel.e; 
{endregion}

{region " SIGNAL AREA : NAME->S_Pnt_Chrg_Mode LENGTH->2 STARTBIT :18"}
_FB_CanTx_Message_Unpack_4A0.S_Bit_18		:= (GVL.IOVD.S_Pnt_Chrg_Mode.x OR GVL.IOVD.S_Pnt_Chrg_Mode.na) AND NOT GVL.IOVD.S_Pnt_Chrg_Mode.e; 
_FB_CanTx_Message_Unpack_4A0.S_Bit_19		:= NOT GVL.IOVD.S_Pnt_Chrg_Mode.v OR GVL.IOVD.S_Pnt_Chrg_Mode.na OR GVL.IOVD.S_Pnt_Chrg_Mode.e; 
{endregion}

{region " SIGNAL AREA : NAME->S_TCU_Pnt_Chrg_Ct LENGTH->2 STARTBIT :20"}
_FB_CanTx_Message_Unpack_4A0.S_Bit_20		:= (GVL.IOVD.S_TCU_Pnt_Chrg_Ct.x OR GVL.IOVD.S_TCU_Pnt_Chrg_Ct.na) AND NOT GVL.IOVD.S_TCU_Pnt_Chrg_Ct.e; 
_FB_CanTx_Message_Unpack_4A0.S_Bit_21		:= NOT GVL.IOVD.S_TCU_Pnt_Chrg_Ct.v OR GVL.IOVD.S_TCU_Pnt_Chrg_Ct.na OR GVL.IOVD.S_TCU_Pnt_Chrg_Ct.e; 
{endregion}

{region " SIGNAL AREA : NAME->S_TCU_Chrg_Ct LENGTH->2 STARTBIT :22"}
_FB_CanTx_Message_Unpack_4A0.S_Bit_22		:= (GVL.IOVD.S_TCU_Chrg_Ct.x OR GVL.IOVD.S_TCU_Chrg_Ct.na) AND NOT GVL.IOVD.S_TCU_Chrg_Ct.e; 
_FB_CanTx_Message_Unpack_4A0.S_Bit_23		:= NOT GVL.IOVD.S_TCU_Chrg_Ct.v OR GVL.IOVD.S_TCU_Chrg_Ct.na OR GVL.IOVD.S_TCU_Chrg_Ct.e; 
{endregion}

_FB_CanTx_Message_Unpack_4A0.S_Bit_6			:= TRUE;
_FB_CanTx_Message_Unpack_4A0.S_Bit_7			:= TRUE;
_FB_CanTx_Message_Unpack_4A0.S_Bit_14			:= TRUE;
_FB_CanTx_Message_Unpack_4A0.S_Bit_15			:= TRUE;
_FB_CanTx_Message_Unpack_4A0.X_Byte_3			:= 16#FF;
_FB_CanTx_Message_Unpack_4A0.S_Bit_32			:= TRUE;
_FB_CanTx_Message_Unpack_4A0.S_Bit_33			:= TRUE;
_FB_CanTx_Message_Unpack_4A0.S_Bit_34			:= TRUE;
_FB_CanTx_Message_Unpack_4A0.S_Bit_35			:= TRUE;
_FB_CanTx_Message_Unpack_4A0.S_Bit_36			:= TRUE;
_FB_CanTx_Message_Unpack_4A0.S_Bit_37			:= TRUE;
_FB_CanTx_Message_Unpack_4A0.S_Bit_38			:= TRUE;
_FB_CanTx_Message_Unpack_4A0.S_Bit_39			:= TRUE;
_FB_CanTx_Message_Unpack_4A0.X_Byte_5			:= 16#FF;
_FB_CanTx_Message_Unpack_4A0.X_Byte_6			:= 16#FF;
_FB_CanTx_Message_Unpack_4A0.X_Byte_7			:= 16#FF;

_FB_CanTx_Message_Unpack_4A0 (		C_Enable		:= GVL.IOVD.C_En_Sarj_Durum_0X4A0,
     								Obj_CAN			:= ADR(GVL.IC.Obj_CAN0),
     								X_MsgID			:= 16#4A0,
     								Tm_CycleTime	:= TIME#500MS,
     								N_Msg_Dlc		:= 8,
     								S_Extended		:= 0,
     								S_Sent_Ok   	=> GVL.IOVD.S_SentOk_Sarj_Durum_0X4A0);
{endregion}
//-----------------------------------------------------------------------------------------------------------------------------
//-----------------------------------------------------------------------------------------------------------------------------
{region " MESSAGE AREA :Sarj_Sureleri- ID:4A5"}

{region " SIGNAL AREA : NAME->X_Tm_Seri_Hour LENGTH->8 STARTBIT :0"}
_FB_CanTx_Message_Unpack_4A5.X_Byte_0					:=
(*SELECT 1 : Is data valid and range is not exceed?*)	SEL((GVL.IOVD.X_Tm_Seri_Hour.v AND NOT GVL.IOVD.X_Tm_Seri_Hour.RangeExcd),
(*SELECT 2 : Is NOT AVAILABLE ?*)						SEL(GVL.IOVD.X_Tm_Seri_Hour.na,
(*SELECT 3 : Is ERROR active ?*)						SEL(GVL.IOVD.X_Tm_Seri_Hour.e,
(*DEFAULT VALUE assignment*)							0,
(*ERROR is active*)										16#FE),
(*NOT AVAILABLE is active*)								16#FF),
(*Transmission is VALID*)								USINT_TO_BYTE(REAL_TO_USINT((GVL.IOVD.X_Tm_Seri_Hour.x))));
{endregion}

{region " SIGNAL AREA : NAME->X_Tm_Seri_Minute LENGTH->8 STARTBIT :8"}
_FB_CanTx_Message_Unpack_4A5.X_Byte_1					:=
(*SELECT 1 : Is data valid and range is not exceed?*)	SEL((GVL.IOVD.X_Tm_Seri_Minute.v AND NOT GVL.IOVD.X_Tm_Seri_Minute.RangeExcd),
(*SELECT 2 : Is NOT AVAILABLE ?*)						SEL(GVL.IOVD.X_Tm_Seri_Minute.na,
(*SELECT 3 : Is ERROR active ?*)						SEL(GVL.IOVD.X_Tm_Seri_Minute.e,
(*DEFAULT VALUE assignment*)							0,
(*ERROR is active*)										16#FE),
(*NOT AVAILABLE is active*)								16#FF),
(*Transmission is VALID*)								USINT_TO_BYTE(REAL_TO_USINT((GVL.IOVD.X_Tm_Seri_Minute.x))));
{endregion}

{region " SIGNAL AREA : NAME->X_Tm_Sp_Mode_Hour LENGTH->8 STARTBIT :32"}
_FB_CanTx_Message_Unpack_4A5.X_Byte_4					:=
(*SELECT 1 : Is data valid and range is not exceed?*)	SEL((GVL.IOVD.X_Tm_Sp_Mode_Hour.v AND NOT GVL.IOVD.X_Tm_Sp_Mode_Hour.RangeExcd),
(*SELECT 2 : Is NOT AVAILABLE ?*)						SEL(GVL.IOVD.X_Tm_Sp_Mode_Hour.na,
(*SELECT 3 : Is ERROR active ?*)						SEL(GVL.IOVD.X_Tm_Sp_Mode_Hour.e,
(*DEFAULT VALUE assignment*)							0,
(*ERROR is active*)										16#FE),
(*NOT AVAILABLE is active*)								16#FF),
(*Transmission is VALID*)								USINT_TO_BYTE(REAL_TO_USINT((GVL.IOVD.X_Tm_Sp_Mode_Hour.x))));
{endregion}

{region " SIGNAL AREA : NAME->X_Tm_Sp_Mode_Minute LENGTH->8 STARTBIT :40"}
_FB_CanTx_Message_Unpack_4A5.X_Byte_5					:=
(*SELECT 1 : Is data valid and range is not exceed?*)	SEL((GVL.IOVD.X_Tm_Sp_Mode_Minute.v AND NOT GVL.IOVD.X_Tm_Sp_Mode_Minute.RangeExcd),
(*SELECT 2 : Is NOT AVAILABLE ?*)						SEL(GVL.IOVD.X_Tm_Sp_Mode_Minute.na,
(*SELECT 3 : Is ERROR active ?*)						SEL(GVL.IOVD.X_Tm_Sp_Mode_Minute.e,
(*DEFAULT VALUE assignment*)							0,
(*ERROR is active*)										16#FE),
(*NOT AVAILABLE is active*)								16#FF),
(*Transmission is VALID*)								USINT_TO_BYTE(REAL_TO_USINT((GVL.IOVD.X_Tm_Sp_Mode_Minute.x))));
{endregion}

{region " SIGNAL AREA : NAME->X_Tm_Estm_Fn_Hour LENGTH->8 STARTBIT :48"}
_FB_CanTx_Message_Unpack_4A5.X_Byte_6					:=
(*SELECT 1 : Is data valid and range is not exceed?*)	SEL((GVL.IOVD.X_Tm_Estm_Fn_Hour.v AND NOT GVL.IOVD.X_Tm_Estm_Fn_Hour.RangeExcd),
(*SELECT 2 : Is NOT AVAILABLE ?*)						SEL(GVL.IOVD.X_Tm_Estm_Fn_Hour.na,
(*SELECT 3 : Is ERROR active ?*)						SEL(GVL.IOVD.X_Tm_Estm_Fn_Hour.e,
(*DEFAULT VALUE assignment*)							0,
(*ERROR is active*)										16#FE),
(*NOT AVAILABLE is active*)								16#FF),
(*Transmission is VALID*)								USINT_TO_BYTE(REAL_TO_USINT((GVL.IOVD.X_Tm_Estm_Fn_Hour.x))));
{endregion}

{region " SIGNAL AREA : NAME->X_Tm_Estm_Fn_Minute LENGTH->8 STARTBIT :56"}
_FB_CanTx_Message_Unpack_4A5.X_Byte_7					:=
(*SELECT 1 : Is data valid and range is not exceed?*)	SEL((GVL.IOVD.X_Tm_Estm_Fn_Minute.v AND NOT GVL.IOVD.X_Tm_Estm_Fn_Minute.RangeExcd),
(*SELECT 2 : Is NOT AVAILABLE ?*)						SEL(GVL.IOVD.X_Tm_Estm_Fn_Minute.na,
(*SELECT 3 : Is ERROR active ?*)						SEL(GVL.IOVD.X_Tm_Estm_Fn_Minute.e,
(*DEFAULT VALUE assignment*)							0,
(*ERROR is active*)										16#FE),
(*NOT AVAILABLE is active*)								16#FF),
(*Transmission is VALID*)								USINT_TO_BYTE(REAL_TO_USINT((GVL.IOVD.X_Tm_Estm_Fn_Minute.x))));
{endregion}

_FB_CanTx_Message_Unpack_4A5.X_Byte_2				:= 16#FF;
_FB_CanTx_Message_Unpack_4A5.X_Byte_3				:= 16#FF;

_FB_CanTx_Message_Unpack_4A5 (		C_Enable		:= GVL.IOVD.C_En_Sarj_Sureleri_0X4A5,
     								Obj_CAN			:= ADR(GVL.IC.Obj_CAN0),
     								X_MsgID			:= 16#4A5,
     								Tm_CycleTime	:= TIME#500MS,
     								N_Msg_Dlc		:= 8,
     								S_Extended		:= 0,
     								S_Sent_Ok   	=> GVL.IOVD.S_SentOk_Sarj_Sureleri_0X4A5);
{endregion}
//-----------------------------------------------------------------------------------------------------------------------------
//-----------------------------------------------------------------------------------------------------------------------------
{region " MESSAGE AREA :Sarj_Durum_3- ID:4A6"}

// PR1006_SRS_001099_TIMTRO
// PR1006_SRS_001102_TIMTRO
// PR1006_SRS_001100_TIMTRO
{region " SIGNAL AREA : NAME->Z_Ext_Chrg_Stat LENGTH->8 STARTBIT :0"}
_FB_CanTx_Message_Unpack_4A6.X_Byte_0					:=
(*SELECT 1 : Is data valid and range is not exceed?*)	SEL((GVL.IOVD.Z_Ext_Chrg_Stat.v AND NOT GVL.IOVD.Z_Ext_Chrg_Stat.RangeExcd),
(*SELECT 2 : Is NOT AVAILABLE ?*)						SEL(GVL.IOVD.Z_Ext_Chrg_Stat.na,
(*SELECT 3 : Is ERROR active ?*)						SEL(GVL.IOVD.Z_Ext_Chrg_Stat.e,
(*DEFAULT VALUE assignment*)							0,
(*ERROR is active*)										16#E),
(*NOT AVAILABLE is active*)								16#F),
(*Transmission is VALID*)								GVL.IOVD.Z_Ext_Chrg_Stat.x);
{endregion}

{region " SIGNAL AREA : NAME->Z_Pan_Chrg_Stat LENGTH->8 STARTBIT :8"}
_FB_CanTx_Message_Unpack_4A6.X_Byte_1					:=
(*SELECT 1 : Is data valid and range is not exceed?*)	SEL((GVL.IOVD.Z_Pan_Chrg_Stat.v AND NOT GVL.IOVD.Z_Pan_Chrg_Stat.RangeExcd),
(*SELECT 2 : Is NOT AVAILABLE ?*)						SEL(GVL.IOVD.Z_Pan_Chrg_Stat.na,
(*SELECT 3 : Is ERROR active ?*)						SEL(GVL.IOVD.Z_Pan_Chrg_Stat.e,
(*DEFAULT VALUE assignment*)							0,
(*ERROR is active*)										16#E),
(*NOT AVAILABLE is active*)								16#F),
(*Transmission is VALID*)								GVL.IOVD.Z_Pan_Chrg_Stat.x);
{endregion}

{region " SIGNAL AREA : NAME->Z_Pnt_Pos LENGTH->8 STARTBIT :16"}
_FB_CanTx_Message_Unpack_4A6.X_Byte_2					:=
(*SELECT 1 : Is data valid and range is not exceed?*)	SEL((GVL.IOVD.Z_Pnt_Pos.v AND NOT GVL.IOVD.Z_Pnt_Pos.RangeExcd),
(*SELECT 2 : Is NOT AVAILABLE ?*)						SEL(GVL.IOVD.Z_Pnt_Pos.na,
(*SELECT 3 : Is ERROR active ?*)						SEL(GVL.IOVD.Z_Pnt_Pos.e,
(*DEFAULT VALUE assignment*)							0,
(*ERROR is active*)										16#E),
(*NOT AVAILABLE is active*)								16#F),
(*Transmission is VALID*)								GVL.IOVD.Z_Pnt_Pos.x);
{endregion}

_FB_CanTx_Message_Unpack_4A6.X_Byte_3	 :=	16#FF;
_FB_CanTx_Message_Unpack_4A6.X_Byte_4	 :=	16#FF;
_FB_CanTx_Message_Unpack_4A6.X_Byte_5	 :=	16#FF;
_FB_CanTx_Message_Unpack_4A6.X_Byte_6	 :=	16#FF;
_FB_CanTx_Message_Unpack_4A6.X_Byte_7	 :=	16#FF;
	 
_FB_CanTx_Message_Unpack_4A6 (		C_Enable		:= GVL.IOVD.C_En_Sarj_Durum_3_0X4A6,
     								Obj_CAN			:= ADR(GVL.IC.Obj_CAN0),
     								X_MsgID			:= 16#4A6,
     								Tm_CycleTime	:= TIME#500MS,
     								N_Msg_Dlc		:= 8,
     								S_Extended		:= 0,
     								S_Sent_Ok   	=> GVL.IOVD.S_SentOk_Sarj_Durum_3_0X4A6);
{endregion}
//-----------------------------------------------------------------------------------------------------------------------------
//-----------------------------------------------------------------------------------------------------------------------------
{region " MESSAGE AREA :Pantograph_Analog_4 - ID:4AF"}

{region " SIGNAL AREA : NAME->X_I_Pnt_Chrg LENGTH->16 STARTBIT :0"}
_FB_UNPACK_WORD_TO_BYTE_23 (
		X_WORD_0										:= 
(*SELECT 1 : Is data valid and range is not exceed?*)	SEL((GVL.IOVD.X_I_Pnt_Chrg.v AND NOT GVL.IOVD.X_I_Pnt_Chrg.RangeExcd),
(*SELECT 2 : Is NOT AVAILABLE ?*)						SEL(GVL.IOVD.X_I_Pnt_Chrg.na,
(*SELECT 3 : Is ERROR active ?*)						SEL(GVL.IOVD.X_I_Pnt_Chrg.e,
(*DEFAULT VALUE assignment*)							0,
(*ERROR is active*)										16#FEFE),
(*NOT AVAILABLE is active*)								16#FFFF),
(*Transmission is VALID*)								UINT_TO_WORD(REAL_TO_UINT(((GVL.IOVD.X_I_Pnt_Chrg.x - (-750)) / 0.025)))),
		X_BYTE_0										=> _FB_CanTx_Message_Unpack_4AF.X_Byte_0,
		X_BYTE_1										=> _FB_CanTx_Message_Unpack_4AF.X_Byte_1);
{endregion}

{region " SIGNAL AREA : NAME->X_I_Pnt_Chrg LENGTH->16 STARTBIT :16"}
_FB_UNPACK_WORD_TO_BYTE_24 (
		X_WORD_0										:= 
(*SELECT 1 : Is data valid and range is not exceed?*)	SEL((GVL.IOVD.X_U_Pnt_Chrg.v AND NOT GVL.IOVD.X_U_Pnt_Chrg.RangeExcd),
(*SELECT 2 : Is NOT AVAILABLE ?*)						SEL(GVL.IOVD.X_U_Pnt_Chrg.na,
(*SELECT 3 : Is ERROR active ?*)						SEL(GVL.IOVD.X_U_Pnt_Chrg.e,
(*DEFAULT VALUE assignment*)							0,
(*ERROR is active*)										16#FEFE),
(*NOT AVAILABLE is active*)								16#FFFF),
(*Transmission is VALID*)								UINT_TO_WORD(REAL_TO_UINT((GVL.IOVD.X_U_Pnt_Chrg.x) / 0.025))),
		X_BYTE_0										=> _FB_CanTx_Message_Unpack_4AF.X_Byte_2,
		X_BYTE_1										=> _FB_CanTx_Message_Unpack_4AF.X_Byte_3);
{endregion}

{region " SIGNAL AREA : NAME->X_P_Pnt_Chrg LENGTH->16 STARTBIT :32"}
_FB_UNPACK_WORD_TO_BYTE_25 (
		X_WORD_0										:= 
(*SELECT 1 : Is data valid and range is not exceed?*)	SEL((GVL.IOVD.X_P_Pnt_Chrg.v AND NOT GVL.IOVD.X_P_Pnt_Chrg.RangeExcd),
(*SELECT 2 : Is NOT AVAILABLE ?*)						SEL(GVL.IOVD.X_P_Pnt_Chrg.na,
(*SELECT 3 : Is ERROR active ?*)						SEL(GVL.IOVD.X_P_Pnt_Chrg.e,
(*DEFAULT VALUE assignment*)							0,
(*ERROR is active*)										16#FEFE),
(*NOT AVAILABLE is active*)								16#FFFF),
(*Transmission is VALID*)								UINT_TO_WORD(REAL_TO_UINT((GVL.IOVD.X_P_Pnt_Chrg.x + 3276.6)/0.1))),
		X_BYTE_0										=> _FB_CanTx_Message_Unpack_4AF.X_Byte_4,
		X_BYTE_1										=> _FB_CanTx_Message_Unpack_4AF.X_Byte_5);
{endregion}

{region " SIGNAL AREA : NAME->X_T_Pnt_Chrg LENGTH->8 STARTBIT :48"}
_FB_CanTx_Message_Unpack_4AF.X_Byte_6					:=
(*SELECT 1 : Is data valid and range is not exceed?*)	SEL((GVL.IOVD.X_T_Pnt_Chrg.v AND NOT GVL.IOVD.X_T_Pnt_Chrg.RangeExcd),
(*SELECT 2 : Is NOT AVAILABLE ?*)						SEL(GVL.IOVD.X_T_Pnt_Chrg.na,
(*SELECT 3 : Is ERROR active ?*)						SEL(GVL.IOVD.X_T_Pnt_Chrg.e,
(*DEFAULT VALUE assignment*)							USINT_TO_BYTE(REAL_TO_USINT((40))),
(*ERROR is active*)										16#FE),
(*NOT AVAILABLE is active*)								16#FF),
(*Transmission is VALID*)								USINT_TO_BYTE(REAL_TO_USINT((GVL.IOVD.X_T_Pnt_Chrg.x + 40))));	
{endregion}

_FB_CanTx_Message_Unpack_4AF.X_Byte_7 				:= 16#FF;

_FB_CanTx_Message_Unpack_4AF (		C_Enable		:= GVL.IOVD.C_En_Pantograph_Analog_4_0X4AF,
     								Obj_CAN			:= ADR(GVL.IC.Obj_CAN0),
     								X_MsgID			:= 16#4AF,
     								Tm_CycleTime	:= TIME#500MS,
     								N_Msg_Dlc		:= 8,
     								S_Extended		:= 0,
     								S_Sent_Ok   	=> GVL.IOVD.S_SentOk_Pantograph_Analog_4_0X4AF);
{endregion}
//-----------------------------------------------------------------------------------------------------------------------------
//-----------------------------------------------------------------------------------------------------------------------------
{region " MESSAGE AREA :Hava_Kompresoru_Durum- ID:4F0"}

{region " SIGNAL AREA : NAME->C_Air_Cmp_On LENGTH->2 STARTBIT :0"}
_FB_CanTx_Message_Unpack_4F0.S_Bit_0		:= (GVL.IOVD.C_Air_Cmp_On.x OR GVL.IOVD.C_Air_Cmp_On.na) AND NOT GVL.IOVD.C_Air_Cmp_On.e; 
_FB_CanTx_Message_Unpack_4F0.S_Bit_1		:= NOT GVL.IOVD.C_Air_Cmp_On.v OR GVL.IOVD.C_Air_Cmp_On.na OR GVL.IOVD.C_Air_Cmp_On.e; 

{endregion}

{region " SIGNAL AREA : NAME->S_Air_Cmp_On LENGTH->2 STARTBIT :2"}
_FB_CanTx_Message_Unpack_4F0.S_Bit_2		:= (GVL.IOVD.S_Air_Cmp_On.x OR GVL.IOVD.S_Air_Cmp_On.na) AND NOT GVL.IOVD.S_Air_Cmp_On.e; 
_FB_CanTx_Message_Unpack_4F0.S_Bit_3		:= NOT GVL.IOVD.S_Air_Cmp_On.v OR GVL.IOVD.S_Air_Cmp_On.na OR GVL.IOVD.S_Air_Cmp_On.e; 

{endregion}

{region " SIGNAL AREA : NAME->S_ER_Air_Cmp LENGTH->2 STARTBIT :4"}
_FB_CanTx_Message_Unpack_4F0.S_Bit_4		:= (GVL.IOVD.S_ER_Air_Cmp.x OR GVL.IOVD.S_ER_Air_Cmp.na) AND NOT GVL.IOVD.S_ER_Air_Cmp.e; 
_FB_CanTx_Message_Unpack_4F0.S_Bit_5		:= NOT GVL.IOVD.S_ER_Air_Cmp.v OR GVL.IOVD.S_ER_Air_Cmp.na OR GVL.IOVD.S_ER_Air_Cmp.e; 

{endregion}

{region " SIGNAL AREA : NAME->S_ER_Hi_Temp_Air_Cmp LENGTH->2 STARTBIT :6"}
_FB_CanTx_Message_Unpack_4F0.S_Bit_6		:= (GVL.IOVD.S_ER_Hi_Temp_Air_Cmp.x OR GVL.IOVD.S_ER_Hi_Temp_Air_Cmp.na) AND NOT GVL.IOVD.S_ER_Hi_Temp_Air_Cmp.e; 
_FB_CanTx_Message_Unpack_4F0.S_Bit_7		:= NOT GVL.IOVD.S_ER_Hi_Temp_Air_Cmp.v OR GVL.IOVD.S_ER_Hi_Temp_Air_Cmp.na OR GVL.IOVD.S_ER_Hi_Temp_Air_Cmp.e; 
{endregion}

{region " SIGNAL AREA : NAME->S_ER_Psb_Air_Lek LENGTH->2 STARTBIT :8"}
_FB_CanTx_Message_Unpack_4F0.S_Bit_8		:= (GVL.IOVD.S_ER_Psb_Air_Lek.x OR GVL.IOVD.S_ER_Psb_Air_Lek.na) AND NOT GVL.IOVD.S_ER_Psb_Air_Lek.e; 
_FB_CanTx_Message_Unpack_4F0.S_Bit_9		:= NOT GVL.IOVD.S_ER_Psb_Air_Lek.v OR GVL.IOVD.S_ER_Psb_Air_Lek.na OR GVL.IOVD.S_ER_Psb_Air_Lek.e; 
{endregion}

_FB_CanTx_Message_Unpack_4F0.S_Bit_10 		:= TRUE;
_FB_CanTx_Message_Unpack_4F0.S_Bit_11 		:= TRUE;
_FB_CanTx_Message_Unpack_4F0.S_Bit_12 		:= TRUE;
_FB_CanTx_Message_Unpack_4F0.S_Bit_13 		:= TRUE;
_FB_CanTx_Message_Unpack_4F0.S_Bit_14 		:= TRUE;
_FB_CanTx_Message_Unpack_4F0.S_Bit_15 		:= TRUE;

_FB_CanTx_Message_Unpack_4F0.X_Byte_2 		:= 16#FF;
_FB_CanTx_Message_Unpack_4F0.X_Byte_3 		:= 16#FF;
_FB_CanTx_Message_Unpack_4F0.X_Byte_4 		:= 16#FF;
_FB_CanTx_Message_Unpack_4F0.X_Byte_5 		:= 16#FF;
_FB_CanTx_Message_Unpack_4F0.X_Byte_6 		:= 16#FF;
_FB_CanTx_Message_Unpack_4F0.X_Byte_7 		:= 16#FF;

_FB_CanTx_Message_Unpack_4F0 (		C_Enable		:= GVL.IOVD.C_En_Hava_Kompresoru_Durum_0X4F0,
     								Obj_CAN			:= ADR(GVL.IC.Obj_CAN0),
     								X_MsgID			:= 16#4F0,
     								Tm_CycleTime	:= TIME#500MS,
     								N_Msg_Dlc		:= 8,
     								S_Extended		:= 0,
     								S_Sent_Ok   	=> GVL.IOVD.S_SentOk_Hava_Kompresoru_Durum_0X4F0);
{endregion}
//-----------------------------------------------------------------------------------------------------------------------------
                  
END_PROGRAM

(* PR1006_REV_002446_TIMTRO, Serdar Temeltaşı @19.06.2025 BTMS toplam çalışma süresinin 0x4CB grubundaki N_Btms_Op_Cnt sinyali ile DIAG CAN'e gönderilmesi sağlandı. PR1006_REV_002519_TIMTRO, Serdar Temeltaşı @20.06.2025 Hesaplanan hava kompresörü çalışma süresi DIAG CAN'e 0x4CC grubunda gönderildi. PR1006_REV_002637_TIMTRO, Serdar Temeltaşı @08.07.2025 Klima toplam kullanım süresi, sürücü kliması toplam çalışma süresi ve yolcu kliması toplam çalışma süresi değerleri saat cinsinden DWP'ye gönderildi. PR1006_REV_002702_TIMTRO, Serdar Temeltaşı @10.07.2025 DWP'ye gönderilen araçtan ayrılış, 1.kapı üstü led aydınlatma süresi ve validatör kapanma süresi değerlerinin çözünürlüğü 5 olarak değiştirildi. *)
PROGRAM P_IOVD_C
  VAR
    _FB_CanTx_Message_Unpack_403 : _FB_CanTx_Message_Unpack;
    _FB_CanTx_Message_Unpack_410 : _FB_CanTx_Message_Unpack;
    _FB_CanTx_Message_411 : _FB_CanTx_Message;
    _FB_CanTx_Message_413 : _FB_CanTx_Message;
    _FB_CanTx_Message_Unpack_414 : _FB_CanTx_Message_Unpack;
    _FB_CanTx_Message_Unpack_415 : _FB_CanTx_Message_Unpack;
    _FB_CanTx_Message_Unpack_416 : _FB_CanTx_Message_Unpack;
    _FB_CanTx_Message_4C0 : _FB_CanTx_Message;
    _FB_CanTx_Message_4C1 : _FB_CanTx_Message;
    _FB_CanTx_Message_4C3 : _FB_CanTx_Message;
    _FB_CanTx_Message_4C4 : _FB_CanTx_Message;
    _FB_CanTx_Message_4C5 : _FB_CanTx_Message;
    _FB_CanTx_Message_4C6 : _FB_CanTx_Message;
    _FB_CanTx_Message_4C7 : _FB_CanTx_Message;
    _FB_CanTx_Message_4C8 : _FB_CanTx_Message;
    _FB_CanTx_Message_4C9 : _FB_CanTx_Message;
    _FB_CanTx_Message_4CA : _FB_CanTx_Message;
    _FB_CanTx_Message_4CB : _FB_CanTx_Message;
    _FB_CanTx_Message_Unpack_4CC : _FB_CanTx_Message_Unpack;
    _FB_CanTx_Message_Unpack_4CD : _FB_CanTx_Message_Unpack;
    _FB_CanTx_Message_4E0 : _FB_CanTx_Message;
    _FB_CanTx_Message_4CE : _FB_CanTx_Message;
    _FB_CanTx_Message_4CF : _FB_CanTx_Message;
    _FB_CanTx_Message_4D0 : _FB_CanTx_Message;
    _FB_UNPACK_DWORD_TO_BYTE_18 : _FB_UNPACK_DWORD_TO_BYTE;
    _FB_UNPACK_DWORD_TO_BYTE_0 : _FB_UNPACK_DWORD_TO_BYTE;
    _FB_UNPACK_DWORD_TO_BYTE_1 : _FB_UNPACK_DWORD_TO_BYTE;
    _FB_UNPACK_DWORD_TO_BYTE_2 : _FB_UNPACK_DWORD_TO_BYTE;
    _FB_UNPACK_DWORD_TO_BYTE_3 : _FB_UNPACK_DWORD_TO_BYTE;
    _FB_UNPACK_DWORD_TO_BYTE_4 : _FB_UNPACK_DWORD_TO_BYTE;
    _FB_UNPACK_DWORD_TO_BYTE_5 : _FB_UNPACK_DWORD_TO_BYTE;
    _FB_UNPACK_DWORD_TO_BYTE_6 : _FB_UNPACK_DWORD_TO_BYTE;
    _FB_UNPACK_DWORD_TO_BYTE_7 : _FB_UNPACK_DWORD_TO_BYTE;
    _FB_UNPACK_DWORD_TO_BYTE_8 : _FB_UNPACK_DWORD_TO_BYTE;
    _FB_UNPACK_DWORD_TO_BYTE_9 : _FB_UNPACK_DWORD_TO_BYTE;
    _FB_UNPACK_DWORD_TO_BYTE_10 : _FB_UNPACK_DWORD_TO_BYTE;
    _FB_UNPACK_DWORD_TO_BYTE_11 : _FB_UNPACK_DWORD_TO_BYTE;
    _FB_UNPACK_DWORD_TO_BYTE_12 : _FB_UNPACK_DWORD_TO_BYTE;
    _FB_UNPACK_DWORD_TO_BYTE_13 : _FB_UNPACK_DWORD_TO_BYTE;
    _FB_UNPACK_DWORD_TO_BYTE_14 : _FB_UNPACK_DWORD_TO_BYTE;
    _FB_UNPACK_DWORD_TO_BYTE_15 : _FB_UNPACK_DWORD_TO_BYTE;
    _FB_UNPACK_DWORD_TO_BYTE_16 : _FB_UNPACK_DWORD_TO_BYTE;
    _FB_UNPACK_DWORD_TO_BYTE_17 : _FB_UNPACK_DWORD_TO_BYTE;
    _FB_UNPACK_WORD_TO_BYTE_4 : _FB_UNPACK_WORD_TO_BYTE;
    _FB_UNPACK_WORD_TO_BYTE_5 : _FB_UNPACK_WORD_TO_BYTE;
    _FB_UNPACK_WORD_TO_BYTE_6 : _FB_UNPACK_WORD_TO_BYTE;
    _FB_UNPACK_WORD_TO_BYTE_7 : _FB_UNPACK_WORD_TO_BYTE;
    _FB_UNPACK_WORD_TO_BYTE_8 : _FB_UNPACK_WORD_TO_BYTE;
    _FB_UNPACK_WORD_TO_BYTE_9 : _FB_UNPACK_WORD_TO_BYTE;
    _FB_UNPACK_WORD_TO_BYTE_10 : _FB_UNPACK_WORD_TO_BYTE;
    _FB_UNPACK_WORD_TO_BYTE_11 : _FB_UNPACK_WORD_TO_BYTE;
    _FB_UNPACK_WORD_TO_BYTE_12 : _FB_UNPACK_WORD_TO_BYTE;
    _FB_UNPACK_WORD_TO_BYTE_13 : _FB_UNPACK_WORD_TO_BYTE;
    _FB_UNPACK_WORD_TO_BYTE_14 : _FB_UNPACK_WORD_TO_BYTE;
    _FB_UNPACK_DWORD_TO_BYTE_19 : _FB_UNPACK_DWORD_TO_BYTE;
    _FB_UNPACK_DWORD_TO_BYTE_20 : _FB_UNPACK_DWORD_TO_BYTE;
    _FB_UNPACK_DWORD_TO_BYTE_21 : _FB_UNPACK_DWORD_TO_BYTE;
    _FB_UNPACK_DWORD_TO_BYTE_22 : _FB_UNPACK_DWORD_TO_BYTE;
    _FB_UNPACK_DWORD_TO_BYTE_23 : _FB_UNPACK_DWORD_TO_BYTE;
    _FB_UNPACK_DWORD_TO_BYTE_24 : _FB_UNPACK_DWORD_TO_BYTE;
    _FB_UNPACK_WORD_TO_BYTE_0 : _FB_UNPACK_WORD_TO_BYTE;
    _FB_UNPACK_WORD_TO_BYTE_1 : _FB_UNPACK_WORD_TO_BYTE;
    _FB_UNPACK_WORD_TO_BYTE_2 : _FB_UNPACK_WORD_TO_BYTE;
    _FB_UNPACK_WORD_TO_BYTE_3 : _FB_UNPACK_WORD_TO_BYTE;
    _FB_UNPACK_BYTE_TO_8BITS_0 : _FB_UNPACK_BYTE_TO_8BITS;
    _FB_UNPACK_BYTE_TO_8BITS_1 : _FB_UNPACK_BYTE_TO_8BITS;
    _FB_UNPACK_BYTE_TO_8BITS_2 : _FB_UNPACK_BYTE_TO_8BITS;
    _FB_UNPACK_BYTE_TO_8BITS_3 : _FB_UNPACK_BYTE_TO_8BITS;
    _FB_UNPACK_BYTE_TO_8BITS_4 : _FB_UNPACK_BYTE_TO_8BITS;
    _FB_UNPACK_BYTE_TO_8BITS_5 : _FB_UNPACK_BYTE_TO_8BITS;
    _FB_UNPACK_BYTE_TO_8BITS_6 : _FB_UNPACK_BYTE_TO_8BITS;
    _FB_PACK_8BITS_TO_BYTE_0 : _FB_PACK_8BITS_TO_BYTE;
    _FB_PACK_8BITS_TO_BYTE_1 : _FB_PACK_8BITS_TO_BYTE;
    _FB_PACK_8BITS_TO_BYTE_2 : _FB_PACK_8BITS_TO_BYTE;
    _FB_PACK_8BITS_TO_BYTE_3 : _FB_PACK_8BITS_TO_BYTE;
    _FB_PACK_8BITS_TO_BYTE_4 : _FB_PACK_8BITS_TO_BYTE;
    T_N_Hvac_Pass2_Op_Cnt : UDINT;
    T_N_Btms_Op_Cnt : UDINT;
    T_X_E_Chrg_Pan : REAL;
    T_X_E_Chrg_Onbrd : REAL;
  END_VAR

                    (*
**********************************************************************
Bozankaya A.Ş.
**********************************************************************
Name					: P_IOVD_C
POU Type				: Program
Created by              : COMMUNICATION INTERFACE GENERATOR V1.1.034(denizcikispc), BZK.
Creation Date 			: 2023-07-11T10:34:22
Modifications			: see version description below


Program Description:This program which is created by automatically by communication interface generator 
 handles the TX (OUTPUT) can messages according to CAN_500_LIB 
*********************************************************************

Version 1	
*********************************************************************
Version Description:
- initial version
*********************************************************************
*)
//-----------------------------------------------------------------------------------------------------------------------------
//-----------------------------------------------------------------------------------------------------------------------------
//MESSAGE------
{region " User Area : ECU Parametre- ID:403"}
//-------SIGNAL -> S_ER_Susp_Amb Max: 1 Min: 0 Def: 0 Resolution: 1 Offset: 0
GVL.IOVD.S_ER_Susp_Amb						:= 	(GVL.DM1_Susp.gAmberWarningLampStat = 1 OR GVL.DM1_Susp.gFlashAmberWarningLamp = 1) 
												AND ((GVL.DM1_Err_Log_Susp.gDM1Errors.ui8NrActiveError = 1
												AND GVL.DM1_Err_Log_Susp.gDM1Errors.asErrorDm1[0].ui32Spn <> 62 
												AND GVL.DM1_Err_Log_Susp.gDM1Errors.asErrorDm1[1].ui32Spn <> 62 
												AND GVL.DM1_Err_Log_Susp.gDM1Errors.asErrorDm1[2].ui32Spn <> 62 
												AND GVL.DM1_Err_Log_Susp.gDM1Errors.asErrorDm1[3].ui32Spn <> 62 
												AND GVL.DM1_Err_Log_Susp.gDM1Errors.asErrorDm1[4].ui32Spn <> 62 
												AND GVL.DM1_Err_Log_Susp.gDM1Errors.asErrorDm1[5].ui32Spn <> 62) OR GVL.DM1_Err_Log_Susp.gDM1Errors.ui8NrActiveError > 1);
//-------SIGNAL -> S_ER_Susp_Red Max: 1 Min: 0 Def: 0 Resolution: 1 Offset: 0
GVL.IOVD.S_ER_Susp_Red						:= (GVL.DM1_Susp.gRedStopLampStat = 1 OR GVL.DM1_Susp.gMalfunctionIndicatuorLampStat = 1 OR GVL.DM1_Susp.gFlashRedStopLamp = 1 OR GVL.DM1_Susp.gFlashMalfunctionIndicatorLamp = 1);	 
//-------SIGNAL -> S_ER_Lo_Pr_Amb Max: 1 Min: 0 Def: 0 Resolution: 1 Offset: 0
GVL.IOVD.S_ER_Lo_Pr_Amb						:= GVL.XC.S_ER_Lo_Pr_Amb;
//-------SIGNAL -> S_ER_Lo_Pr_Amb Max: 1 Min: 0 Def: 0 Resolution: 1 Offset: 0
GVL.IOVD.S_ER_Lo_Pr_Red						:= GVL.XC.S_ER_Lo_Pr_Red;	
//-------SIGNAL -> S_ER_Ret Max: 1 Min: 0 Def: 0 Resolution: 1 Offset: 0
GVL.IOVD.S_ER_Ret							:= GVL.EDG.S_ER_Ret;
//-------SIGNAL -> P_X_Tm_Dr_Cl_Rls Max: 250 Min: 0 Def: 0 Resolution: 1 Offset: 0
GVL.IOVD.P_X_Tm_Dr_Cl_Rls.v					:= GVL.SY.S_ECU_Rdy AND NOT GVL.IOVD.P_X_Tm_Dr_Cl_Rls.na AND NOT GVL.IOVD.P_X_Tm_Dr_Cl_Rls.e AND NOT GVL.IOVD.P_X_Tm_Dr_Cl_Rls.RangeExcd;
GVL.IOVD.P_X_Tm_Dr_Cl_Rls.x					:= GVL.Param[Param_E.P_X_Tm_Dr_Cl_Rls].X_Val;
GVL.IOVD.P_X_Tm_Dr_Cl_Rls.e					:= FALSE;
GVL.IOVD.P_X_Tm_Dr_Cl_Rls.na				:= GVL.IIVD.S_TmOut_Parametre_1_0X263;
GVL.IOVD.P_X_Tm_Dr_Cl_Rls.RangeExcd			:= (250 < GVL.IOVD.P_X_Tm_Dr_Cl_Rls.x) OR (0 > GVL.IOVD.P_X_Tm_Dr_Cl_Rls.x);
//-------SIGNAL -> P_X_Tm_Vld_ShtDn Max: 250 Min: 0 Def: 0 Resolution: 1 Offset: 0
GVL.IOVD.P_X_Tm_Vld_ShtDn.v					:= GVL.SY.S_ECU_Rdy AND NOT GVL.IOVD.P_X_Tm_Vld_ShtDn.na AND NOT GVL.IOVD.P_X_Tm_Vld_ShtDn.e AND NOT GVL.IOVD.P_X_Tm_Vld_ShtDn.RangeExcd;
GVL.IOVD.P_X_Tm_Vld_ShtDn.x					:= GVL.Param[Param_E.P_X_Tm_Vld_ShtDn].X_Val;
GVL.IOVD.P_X_Tm_Vld_ShtDn.e					:= FALSE;
GVL.IOVD.P_X_Tm_Vld_ShtDn.na				:= GVL.IIVD.S_TmOut_Parametre_1_0X263;
GVL.IOVD.P_X_Tm_Vld_ShtDn.RangeExcd			:= (250 < GVL.IOVD.P_X_Tm_Vld_ShtDn.x) OR (0 > GVL.IOVD.P_X_Tm_Vld_ShtDn.x);
//-------SIGNAL -> P_X_Tm_Lgt_Dr_ShtDn Max: 250 Min: 0 Def: 0 Resolution: 1 Offset: 0
GVL.IOVD.P_X_Tm_Lgt_Dr_ShtDn.v				:= GVL.SY.S_ECU_Rdy AND NOT GVL.IOVD.P_X_Tm_Lgt_Dr_ShtDn.na AND NOT GVL.IOVD.P_X_Tm_Lgt_Dr_ShtDn.e AND NOT GVL.IOVD.P_X_Tm_Lgt_Dr_ShtDn.RangeExcd;
GVL.IOVD.P_X_Tm_Lgt_Dr_ShtDn.x				:= GVL.Param[Param_E.P_X_Tm_Lgt_Dr_ShtDn].X_Val;
GVL.IOVD.P_X_Tm_Lgt_Dr_ShtDn.e				:= FALSE;
GVL.IOVD.P_X_Tm_Lgt_Dr_ShtDn.na				:= GVL.IIVD.S_TmOut_Parametre_1_0X263;
GVL.IOVD.P_X_Tm_Lgt_Dr_ShtDn.RangeExcd		:= (250 < GVL.IOVD.P_X_Tm_Lgt_Dr_ShtDn.x) OR (0 > GVL.IOVD.P_X_Tm_Lgt_Dr_ShtDn.x);
{endregion}
//-----------------------------------------------------------------------------------------------------------------------------
//-----------------------------------------------------------------------------------------------------------------------------
//MESSAGE------
{region " User Area : HVAC_Durum- ID:410"}
//-------SIGNAL -> S_HVAC_Sp Max: 1 Min: 0 Def: 0 Resolution: 1 Offset: 0
GVL.IOVD.S_HVAC_Sp.v							:= GVL.SY.S_ECU_Rdy AND NOT GVL.IOVD.S_HVAC_Sp.e AND NOT GVL.IOVD.S_HVAC_Sp.na;
GVL.IOVD.S_HVAC_Sp.x							:= GVL.MR.S_B2_On;
GVL.IOVD.S_HVAC_Sp.e							:= FALSE;
GVL.IOVD.S_HVAC_Sp.na							:= FALSE;
//-------SIGNAL -> S_HVAC_Mn_Swc Max: 1 Min: 0 Def: 0 Resolution: 1 Offset: 0
GVL.IOVD.S_HVAC_Mn_Swc.v						:= GVL.SY.S_ECU_Rdy AND NOT GVL.IOVD.S_HVAC_Mn_Swc.e AND NOT GVL.IOVD.S_HVAC_Mn_Swc.na;
GVL.IOVD.S_HVAC_Mn_Swc.x						:= GVL.IICH.S_Mn_Swc_Actv.x;
GVL.IOVD.S_HVAC_Mn_Swc.e						:= GVL.IICH.S_Mn_Swc_Actv.e;
GVL.IOVD.S_HVAC_Mn_Swc.na						:= GVL.IICH.S_Mn_Swc_Actv.na;
//-------SIGNAL -> S_HVAC_Otp_Do Max: 1 Min: 0 Def: 0 Resolution: 1 Offset: 0
GVL.IOVD.S_HVAC_Otp_Do.v						:= GVL.SY.S_ECU_Rdy AND NOT GVL.IOVD.S_HVAC_Otp_Do.e AND NOT GVL.IOVD.S_HVAC_Otp_Do.na;
GVL.IOVD.S_HVAC_Otp_Do.x						:= FALSE;
GVL.IOVD.S_HVAC_Otp_Do.e						:= FALSE;
GVL.IOVD.S_HVAC_Otp_Do.na						:= TRUE;
//-------SIGNAL -> C_Dmst_On Max: 1 Min: 0 Def: 0 Resolution: 1 Offset: 0
GVL.IOVD.C_Dmst_On.v							:= GVL.SY.S_ECU_Rdy AND NOT GVL.IOVD.C_Dmst_On.e AND NOT GVL.IOVD.C_Dmst_On.na;
GVL.IOVD.C_Dmst_On.x							:= GVL.CH.C_Dmst_On;
GVL.IOVD.C_Dmst_On.e							:= FALSE;
GVL.IOVD.C_Dmst_On.na							:= FALSE; // GVL.IICH.S_Com_Flt
//-------SIGNAL -> S_BTMS_En Max: 1 Min: 0 Def: 0 Resolution: 1 Offset: 0
GVL.IOVD.S_BTMS_En.v							:= GVL.SY.S_ECU_Rdy AND NOT GVL.IOVD.S_BTMS_En.e AND NOT GVL.IOVD.S_BTMS_En.na;
GVL.IOVD.S_BTMS_En.x							:= GVL.IICH.Z_BTMS.x <> 0;
GVL.IOVD.S_BTMS_En.e							:= GVL.IICH.Z_BTMS.e;
GVL.IOVD.S_BTMS_En.na							:= GVL.IICH.Z_BTMS.na;
//-------SIGNAL -> S_Elec_Heat_1_En Max: 1 Min: 0 Def: 0 Resolution: 1 Offset: 0
GVL.IOVD.S_Elec_Heat_1_En.v						:= GVL.SY.S_ECU_Rdy AND NOT GVL.IOVD.S_Elec_Heat_1_En.e AND NOT GVL.IOVD.S_Elec_Heat_1_En.na;
GVL.IOVD.S_Elec_Heat_1_En.x						:= GVL.IICH.C_Elec_Heat_1_On.x;
GVL.IOVD.S_Elec_Heat_1_En.e						:= GVL.IICH.C_Elec_Heat_1_On.e;
GVL.IOVD.S_Elec_Heat_1_En.na					:= GVL.IICH.C_Elec_Heat_1_On.na;
//-------SIGNAL -> S_Elec_Heat_2_En Max: 1 Min: 0 Def: 0 Resolution: 1 Offset: 0
GVL.IOVD.S_Elec_Heat_2_En.v						:= GVL.SY.S_ECU_Rdy AND NOT GVL.IOVD.S_Elec_Heat_2_En.e AND NOT GVL.IOVD.S_Elec_Heat_2_En.na;
GVL.IOVD.S_Elec_Heat_2_En.x						:= GVL.IICH.C_Elec_Heat_2_On.x;
GVL.IOVD.S_Elec_Heat_2_En.e						:= GVL.IICH.C_Elec_Heat_2_On.e;
GVL.IOVD.S_Elec_Heat_2_En.na					:= GVL.IICH.C_Elec_Heat_2_On.na;
//-------SIGNAL -> S_HVAC_Inver_En Max: 1 Min: 0 Def: 0 Resolution: 1 Offset: 0
GVL.IOVD.S_HVAC_Inver_En.v						:= GVL.SY.S_ECU_Rdy AND NOT GVL.IOVD.S_HVAC_Inver_En.e AND NOT GVL.IOVD.S_HVAC_Inver_En.na;
GVL.IOVD.S_HVAC_Inver_En.x						:= GVL.IICH.C_Inv_On.x;
GVL.IOVD.S_HVAC_Inver_En.e						:= GVL.IICH.C_Inv_On.e;
GVL.IOVD.S_HVAC_Inver_En.na						:= GVL.IICH.C_Inv_On.na;
//-------SIGNAL -> S_HVAC_1_En Max: 1 Min: 0 Def: 0 Resolution: 1 Offset: 0
GVL.IOVD.S_HVAC_1_En.v							:= GVL.SY.S_ECU_Rdy AND NOT GVL.IOVD.S_HVAC_1_En.e AND NOT GVL.IOVD.S_HVAC_1_En.na;
GVL.IOVD.S_HVAC_1_En.x							:= GVL.IICH.Z_Act_Op_Mode.x < 15;
GVL.IOVD.S_HVAC_1_En.e							:= GVL.IICH.Z_Act_Op_Mode.e;
GVL.IOVD.S_HVAC_1_En.na							:= GVL.IICH.Z_Act_Op_Mode.na;
//-------SIGNAL -> S_HVAC_2_En Max: 1 Min: 0 Def: 0 Resolution: 1 Offset: 0
GVL.IOVD.S_HVAC_2_En.v							:= GVL.SY.S_ECU_Rdy AND NOT GVL.IOVD.S_HVAC_2_En.e AND NOT GVL.IOVD.S_HVAC_2_En.na;
GVL.IOVD.S_HVAC_2_En.x							:= FALSE;
GVL.IOVD.S_HVAC_2_En.e							:= FALSE;
GVL.IOVD.S_HVAC_2_En.na							:= TRUE;
//-------SIGNAL -> S_HVAC_Drv_En Max: 1 Min: 0 Def: 0 Resolution: 1 Offset: 0
GVL.IOVD.S_HVAC_Drv_En.v						:= GVL.SY.S_ECU_Rdy AND NOT GVL.IOVD.S_HVAC_Drv_En.e AND NOT GVL.IOVD.S_HVAC_Drv_En.na;
GVL.IOVD.S_HVAC_Drv_En.x						:= GVL.CH.S_HVAC_Drv_On;
GVL.IOVD.S_HVAC_Drv_En.e						:= GVL.IICH.S_Drv_Cool.e OR GVL.IICH.S_Drv_Heat.e OR GVL.IICH.S_Drv_Reheat.e OR GVL.IICH.S_Drv_Ven.e;
GVL.IOVD.S_HVAC_Drv_En.na						:= GVL.IICH.S_Drv_Cool.na OR GVL.IICH.S_Drv_Heat.na OR GVL.IICH.S_Drv_Reheat.na OR GVL.IICH.S_Drv_Ven.na;
//-------SIGNAL -> S_BTMS_Actv Max: 1 Min: 0 Def: 0 Resolution: 1 Offset: 0
GVL.IOVD.S_BTMS_Actv.v							:= GVL.SY.S_ECU_Rdy AND NOT GVL.IOVD.S_BTMS_Actv.e AND NOT GVL.IOVD.S_BTMS_Actv.na;
GVL.IOVD.S_BTMS_Actv.x							:= GVL.IICH.Z_BTMS.x <> 0;
GVL.IOVD.S_BTMS_Actv.e							:= GVL.IICH.Z_BTMS.e;
GVL.IOVD.S_BTMS_Actv.na							:= GVL.IICH.Z_BTMS.na;
//-------SIGNAL -> Z_BTMS_Mode Max: 1 Min: 0 Def: 0 Resolution: 1 Offset: 0
GVL.IOVD.Z_BTMS_Mode.v							:= GVL.SY.S_ECU_Rdy;
GVL.IOVD.Z_BTMS_Mode.x							:= SEL(GVL.IICH.Z_BTMS.x = 0, SEL(GVL.IICH.Z_BTMS.x = 1 OR GVL.IICH.Z_BTMS.x = 3, SEL(GVL.IICH.Z_BTMS.x = 2, 0 (*BTMS hatası*), 2) , 1) , 0); 
//-------SIGNAL -> Z_BTMS_Req_Mode Max: 1 Min: 0 Def: 0 Resolution: 1 Offset: 0
GVL.IOVD.Z_BTMS_Req_Mode.v						:= GVL.SY.S_ECU_Rdy AND NOT GVL.IOVD.Z_BTMS_Req_Mode.e AND NOT GVL.IOVD.Z_BTMS_Req_Mode.na;
GVL.IOVD.Z_BTMS_Req_Mode.x						:= GVL.IICH.Z_BTMS_Req.x;
GVL.IOVD.Z_BTMS_Req_Mode.e						:= GVL.IICH.Z_BTMS_Req.e;
GVL.IOVD.Z_BTMS_Req_Mode.na						:= GVL.IICH.Z_BTMS_Req.na;
//-------SIGNAL -> S_Elec_Heat_1_On Max: 1 Min: 0 Def: 0 Resolution: 1 Offset: 0
GVL.IOVD.S_Elec_Heat_1_On.v						:= GVL.SY.S_ECU_Rdy AND NOT GVL.IOVD.S_Elec_Heat_1_On.e AND NOT GVL.IOVD.S_Elec_Heat_1_On.na;
GVL.IOVD.S_Elec_Heat_1_On.x						:= GVL.IICH.X_P_Elec_Heat.x <> 0;
GVL.IOVD.S_Elec_Heat_1_On.e						:= GVL.IICH.X_P_Elec_Heat.e;
GVL.IOVD.S_Elec_Heat_1_On.na					:= GVL.IICH.X_P_Elec_Heat.na;
//-------SIGNAL -> S_Elec_Heat_2_On Max: 1 Min: 0 Def: 0 Resolution: 1 Offset: 0
GVL.IOVD.S_Elec_Heat_2_On.v						:= GVL.SY.S_ECU_Rdy AND NOT GVL.IOVD.S_Elec_Heat_2_On.e AND NOT GVL.IOVD.S_Elec_Heat_2_On.na;
GVL.IOVD.S_Elec_Heat_2_On.x						:= GVL.IICH.X_P_Elec_Heat.x <> 0;
GVL.IOVD.S_Elec_Heat_2_On.e						:= GVL.IICH.X_P_Elec_Heat.e;
GVL.IOVD.S_Elec_Heat_2_On.na					:= GVL.IICH.X_P_Elec_Heat.na;		  
//-------SIGNAL -> S_HVAC_Inver_On Max: 1 Min: 0 Def: 0 Resolution: 1 Offset: 0
GVL.IOVD.S_HVAC_Inver_On.v						:= GVL.SY.S_ECU_Rdy AND NOT GVL.IOVD.S_HVAC_Inver_On.na AND NOT GVL.IOVD.S_HVAC_Inver_On.e;
GVL.IOVD.S_HVAC_Inver_On.x						:= GVL.IICH.X_P_Inv.x <> 0;
GVL.IOVD.S_HVAC_Inver_On.e						:= GVL.IICH.X_P_Inv.e;
GVL.IOVD.S_HVAC_Inver_On.na						:= GVL.IICH.X_P_Inv.na;
//-------SIGNAL -> S_Elec_Heat_Tm_On Max: 1 Min: 0 Def: 0 Resolution: 1 Offset: 0
GVL.IOVD.S_Elec_Heat_Tm_On.v					:= GVL.SY.S_ECU_Rdy AND NOT GVL.IOVD.S_Elec_Heat_Tm_On.na AND NOT GVL.IOVD.S_Elec_Heat_Tm_On.e;
GVL.IOVD.S_Elec_Heat_Tm_On.x					:= FALSE;
GVL.IOVD.S_Elec_Heat_Tm_On.e					:= FALSE;
GVL.IOVD.S_Elec_Heat_Tm_On.na					:= FALSE;
//-------SIGNAL -> Z_HVAC_1_Mode Max: 10 Min: 0 Def: 0 Resolution: 1 Offset: 0
GVL.IOVD.Z_HVAC_1_Mode.v						:= GVL.SY.S_ECU_Rdy AND NOT GVL.IOVD.Z_HVAC_1_Mode.na AND NOT GVL.IOVD.Z_HVAC_1_Mode.e AND NOT GVL.IOVD.Z_HVAC_1_Mode.RangeExcd;
GVL.IOVD.Z_HVAC_1_Mode.x						:= GVL.IICH.Z_Act_Op_Mode.x;
GVL.IOVD.Z_HVAC_1_Mode.e						:= GVL.IICH.Z_Act_Op_Mode.e;
GVL.IOVD.Z_HVAC_1_Mode.na						:= GVL.IICH.Z_Act_Op_Mode.na;
GVL.IOVD.Z_HVAC_1_Mode.RangeExcd				:=  (10 < GVL.IOVD.Z_HVAC_1_Mode.x )OR (0 > GVL.IOVD.Z_HVAC_1_Mode.x);
//-------SIGNAL -> Z_HVAC_2_Mode Max: 10 Min: 0 Def: 0 Resolution: 1 Offset: 0
GVL.IOVD.Z_HVAC_2_Mode.v						:= GVL.SY.S_ECU_Rdy AND NOT GVL.IOVD.Z_HVAC_2_Mode.na AND NOT GVL.IOVD.Z_HVAC_2_Mode.e AND NOT GVL.IOVD.Z_HVAC_2_Mode.RangeExcd;
GVL.IOVD.Z_HVAC_2_Mode.x						:= 0;
GVL.IOVD.Z_HVAC_2_Mode.e						:= FALSE;
GVL.IOVD.Z_HVAC_2_Mode.na						:= TRUE;
GVL.IOVD.Z_HVAC_2_Mode.RangeExcd				:=  (10 < GVL.IOVD.Z_HVAC_2_Mode.x )OR (0 > GVL.IOVD.Z_HVAC_2_Mode.x);
//-------SIGNAL -> Z_HVAC_Drv_Mode Max: 10 Min: 0 Def: 0 Resolution: 1 Offset: 0
GVL.IOVD.Z_HVAC_Drv_Mode.v						:= GVL.SY.S_ECU_Rdy AND NOT GVL.IOVD.Z_HVAC_Drv_Mode.na AND NOT GVL.IOVD.Z_HVAC_Drv_Mode.e AND NOT GVL.IOVD.Z_HVAC_Drv_Mode.RangeExcd;
GVL.IOVD.Z_HVAC_Drv_Mode.x						:= SEL(GVL.IICH.S_Drv_Ven.x, SEL(GVL.IICH.S_Drv_Heat.x OR GVL.IICH.S_Drv_Reheat.x, SEL(GVL.IICH.S_Drv_Cool.x, 0 , 4) , 2), 1);
GVL.IOVD.Z_HVAC_Drv_Mode.e						:= GVL.IICH.S_Drv_Cool.e OR GVL.IICH.S_Drv_Heat.e OR GVL.IICH.S_Drv_Rcr_Air_Actv.e OR GVL.IICH.S_Drv_Reheat.e OR GVL.IICH.S_Drv_Ven.e;
GVL.IOVD.Z_HVAC_Drv_Mode.na						:= GVL.IICH.S_Drv_Cool.na OR GVL.IICH.S_Drv_Heat.na OR GVL.IICH.S_Drv_Rcr_Air_Actv.na OR GVL.IICH.S_Drv_Reheat.na OR GVL.IICH.S_Drv_Ven.na;
GVL.IOVD.Z_HVAC_Drv_Mode.RangeExcd				:=  (10 < GVL.IOVD.Z_HVAC_Drv_Mode.x )OR (0 > GVL.IOVD.Z_HVAC_Drv_Mode.x);
//-------SIGNAL -> Z_ER_HVAC Max: 10 Min: 0 Def: 0 Resolution: 1 Offset: 0
GVL.IOVD.Z_ER_HVAC.v							:= GVL.SY.S_ECU_Rdy AND NOT GVL.IOVD.Z_ER_HVAC.na AND NOT GVL.IOVD.Z_ER_HVAC.e AND NOT GVL.IOVD.Z_ER_HVAC.RangeExcd;
GVL.IOVD.Z_ER_HVAC.x							:= GVL.IICH.N_Actv_Err.x;
GVL.IOVD.Z_ER_HVAC.e							:= GVL.IICH.N_Actv_Err.e;
GVL.IOVD.Z_ER_HVAC.na							:= GVL.IICH.N_Actv_Err.na;
GVL.IOVD.Z_ER_HVAC.RangeExcd					:=  (10 < GVL.IOVD.Z_ER_HVAC.x )OR (0 > GVL.IOVD.Z_ER_HVAC.x);
//-------SIGNAL -> X_Spd_HVAC_Fan Max: 100 Min: 0 Def: 0 Resolution: 1 Offset: 0
GVL.IOVD.X_Spd_HVAC_Fan.v						:= GVL.SY.S_ECU_Rdy AND NOT GVL.IOVD.X_Spd_HVAC_Fan.na AND NOT GVL.IOVD.X_Spd_HVAC_Fan.e AND NOT GVL.IOVD.X_Spd_HVAC_Fan.RangeExcd;
GVL.IOVD.X_Spd_HVAC_Fan.x						:= GVL.IICH.X_Spd_Fan.x;
GVL.IOVD.X_Spd_HVAC_Fan.e						:= GVL.IICH.X_Spd_Fan.e;
GVL.IOVD.X_Spd_HVAC_Fan.na						:= GVL.IICH.X_Spd_Fan.na;
GVL.IOVD.X_Spd_HVAC_Fan.RangeExcd				:=  (100 < GVL.IOVD.X_Spd_HVAC_Fan.x )OR (0 > GVL.IOVD.X_Spd_HVAC_Fan.x);
{endregion}
//-----------------------------------------------------------------------------------------------------------------------------
//-----------------------------------------------------------------------------------------------------------------------------
//MESSAGE------
{region " User Area : HVAC_Sicaklik- ID:411"}

//-------SIGNAL -> X_T_Drv Max: 100 Min: -40 Def: 0 Resolution: 1 Offset: -40
GVL.IOVD.X_T_Drv.v								:= GVL.SY.S_ECU_Rdy AND NOT GVL.IOVD.X_T_Drv.na AND NOT GVL.IOVD.X_T_Drv.e AND NOT GVL.IOVD.X_T_Drv.RangeExcd;
GVL.IOVD.X_T_Drv.x								:= GVL.IICH.X_T_Drv.x;
GVL.IOVD.X_T_Drv.e								:= GVL.IICH.X_T_Drv.e;
GVL.IOVD.X_T_Drv.na								:= GVL.IICH.X_T_Drv.na;
GVL.IOVD.X_T_Drv.RangeExcd						:=  (100 < GVL.IOVD.X_T_Drv.x )OR (-40 > GVL.IOVD.X_T_Drv.x);
//-------SIGNAL -> W_T_Drv Max: 100 Min: -40 Def: 0 Resolution: 1 Offset: -40
GVL.IOVD.W_T_Drv.v								:= GVL.SY.S_ECU_Rdy AND NOT GVL.IOVD.W_T_Drv.na AND NOT GVL.IOVD.W_T_Drv.e AND NOT GVL.IOVD.W_T_Drv.RangeExcd;
GVL.IOVD.W_T_Drv.x								:= GVL.IICH.W_T_Drv.x;
GVL.IOVD.W_T_Drv.e								:= GVL.IICH.W_T_Drv.e;
GVL.IOVD.W_T_Drv.na								:= GVL.IICH.W_T_Drv.na;
GVL.IOVD.W_T_Drv.RangeExcd						:=  (100 < GVL.IOVD.W_T_Drv.x )OR (-40 > GVL.IOVD.W_T_Drv.x);
//-------SIGNAL -> X_T_Insd_1 Max: 200 Min: -40 Def: 0 Resolution: 1 Offset: -40
GVL.IOVD.X_T_Insd_1.v							:= GVL.SY.S_ECU_Rdy AND NOT GVL.IOVD.X_T_Insd_1.na AND NOT GVL.IOVD.X_T_Insd_1.e AND NOT GVL.IOVD.X_T_Insd_1.RangeExcd;
GVL.IOVD.X_T_Insd_1.x							:= GVL.IICH.X_T_Int.x;
GVL.IOVD.X_T_Insd_1.e							:= GVL.IICH.X_T_Int.e;
GVL.IOVD.X_T_Insd_1.na							:= GVL.IICH.X_T_Int.na;
GVL.IOVD.X_T_Insd_1.RangeExcd					:=  (200 < GVL.IOVD.X_T_Drv.x )OR (-40 > GVL.IOVD.X_T_Drv.x);
//-------SIGNAL -> X_T_Insd_2 Max: 100 Min: -40 Def: 0 Resolution: 1 Offset: -40
GVL.IOVD.X_T_Insd_2.v							:= GVL.SY.S_ECU_Rdy AND NOT GVL.IOVD.X_T_Insd_2.na AND NOT GVL.IOVD.X_T_Insd_2.e AND NOT GVL.IOVD.X_T_Insd_2.RangeExcd;
GVL.IOVD.X_T_Insd_2.x							:= GVL.IICH.X_T_Drv.x;
GVL.IOVD.X_T_Insd_2.e							:= GVL.IICH.X_T_Drv.e;
GVL.IOVD.X_T_Insd_2.na							:= GVL.IICH.X_T_Drv.na;
GVL.IOVD.X_T_Insd_2.RangeExcd					:=  (200 < GVL.IOVD.X_T_Drv.x )OR (-40 > GVL.IOVD.X_T_Drv.x);
//-------SIGNAL -> W_T_HVAC_Psng Max: 100 Min: -40 Def: 0 Resolution: 1 Offset: -40
GVL.IOVD.W_T_HVAC_Psng.v						:= GVL.SY.S_ECU_Rdy AND NOT GVL.IOVD.W_T_HVAC_Psng.na AND NOT GVL.IOVD.W_T_HVAC_Psng.e AND NOT GVL.IOVD.W_T_HVAC_Psng.RangeExcd;
GVL.IOVD.W_T_HVAC_Psng.x						:= GVL.IICH.W_T_Int.x;
GVL.IOVD.W_T_HVAC_Psng.e						:= GVL.IICH.W_T_Int.e;
GVL.IOVD.W_T_HVAC_Psng.na						:= GVL.IICH.W_T_Int.na;
GVL.IOVD.W_T_HVAC_Psng.RangeExcd				:=  (100 < GVL.IOVD.W_T_HVAC_Psng.x )OR (-40 > GVL.IOVD.W_T_HVAC_Psng.x);
//-------SIGNAL -> X_T_Amb Max: 100 Min: -40 Def: 0 Resolution: 1 Offset: -40
GVL.IOVD.X_T_Amb.v								:= GVL.SY.S_ECU_Rdy AND NOT GVL.IOVD.X_T_Amb.na AND NOT GVL.IOVD.X_T_Amb.e AND NOT GVL.IOVD.X_T_Amb.RangeExcd;
GVL.IOVD.X_T_Amb.x								:= GVL.IICH.X_T_Amb.x;
GVL.IOVD.X_T_Amb.e								:= GVL.IICH.X_T_Amb.e;
GVL.IOVD.X_T_Amb.na								:= GVL.IICH.X_T_Amb.na;
GVL.IOVD.X_T_Amb.RangeExcd						:=  (100 < GVL.IOVD.X_T_Amb.x )OR (-40 > GVL.IOVD.X_T_Amb.x);
//-------SIGNAL -> X_T_Clt_Wtr Max: 100 Min: -40 Def: 0 Resolution: 1 Offset: -40
GVL.IOVD.X_T_Clt_Wtr.v							:= GVL.SY.S_ECU_Rdy AND NOT GVL.IOVD.X_T_Clt_Wtr.na AND NOT GVL.IOVD.X_T_Clt_Wtr.e AND NOT GVL.IOVD.X_T_Clt_Wtr.RangeExcd;
GVL.IOVD.X_T_Clt_Wtr.x							:= 0; //EKLENECEK
GVL.IOVD.X_T_Clt_Wtr.e							:= FALSE;
GVL.IOVD.X_T_Clt_Wtr.na							:= TRUE;
GVL.IOVD.X_T_Clt_Wtr.RangeExcd					:=  (100 < GVL.IOVD.X_T_Clt_Wtr.x )OR (-40 > GVL.IOVD.X_T_Clt_Wtr.x);
{endregion}
//-----------------------------------------------------------------------------------------------------------------------------
//-----------------------------------------------------------------------------------------------------------------------------
//MESSAGE------
{region " User Area : HVAC_Analog- ID:413"}

//-------SIGNAL -> X_P_HVAC_Inver Max: 64255 Min: 0 Def: 0 Resolution: 1 Offset: 0
GVL.IOVD.X_P_HVAC_Inver.v					:= GVL.SY.S_ECU_Rdy AND NOT GVL.IOVD.X_P_HVAC_Inver.na AND NOT GVL.IOVD.X_P_HVAC_Inver.e AND NOT GVL.IOVD.X_P_HVAC_Inver.RangeExcd;
GVL.IOVD.X_P_HVAC_Inver.x					:= GVL.IICH.X_P_Inv.x;
GVL.IOVD.X_P_HVAC_Inver.e					:= GVL.IICH.X_P_Inv.e;
GVL.IOVD.X_P_HVAC_Inver.na					:= GVL.IICH.X_P_Inv.na;
GVL.IOVD.X_P_HVAC_Inver.RangeExcd			:=  (64255 < GVL.IOVD.X_P_HVAC_Inver.x )OR (0 > GVL.IOVD.X_P_HVAC_Inver.x);
//-------SIGNAL -> X_P_Elec_Heat Max: 64255 Min: 0 Def: 0 Resolution: 1 Offset: 0
GVL.IOVD.X_P_Elec_Heat.v					:= GVL.SY.S_ECU_Rdy AND NOT GVL.IOVD.X_P_Elec_Heat.na AND NOT GVL.IOVD.X_P_Elec_Heat.e AND NOT GVL.IOVD.X_P_Elec_Heat.RangeExcd;
GVL.IOVD.X_P_Elec_Heat.x					:= GVL.IICH.X_P_Elec_Heat.x;
GVL.IOVD.X_P_Elec_Heat.e					:= GVL.IICH.X_P_Elec_Heat.e;
GVL.IOVD.X_P_Elec_Heat.na					:= GVL.IICH.X_P_Elec_Heat.na;
GVL.IOVD.X_P_Elec_Heat.RangeExcd			:=  (64255 < GVL.IOVD.X_P_Elec_Heat.x )OR (0 > GVL.IOVD.X_P_Elec_Heat.x);
//-------SIGNAL -> X_I_In_HVAC_Inver Max: 3212.75 Min: 0 Def: 0 Resolution: 0.05 Offset: 0
GVL.IOVD.X_I_In_HVAC_Inver.v				:= GVL.SY.S_ECU_Rdy AND NOT GVL.IOVD.X_I_In_HVAC_Inver.na AND NOT GVL.IOVD.X_I_In_HVAC_Inver.e AND NOT GVL.IOVD.X_I_In_HVAC_Inver.RangeExcd;
GVL.IOVD.X_I_In_HVAC_Inver.x				:= GVL.IICH.X_I_Inv.x;
GVL.IOVD.X_I_In_HVAC_Inver.e				:= GVL.IICH.X_I_Inv.e;
GVL.IOVD.X_I_In_HVAC_Inver.na				:= GVL.IICH.X_I_Inv.na;
GVL.IOVD.X_I_In_HVAC_Inver.RangeExcd		:=  (3212.75 < GVL.IOVD.X_I_In_HVAC_Inver.x )OR (0 > GVL.IOVD.X_I_In_HVAC_Inver.x);
//-------SIGNAL -> X_I_In_Elec_Heat Max: 3212.75 Min: 0 Def: 0 Resolution: 0.05 Offset: 0
GVL.IOVD.X_I_In_Elec_Heat.v					:= GVL.SY.S_ECU_Rdy AND NOT GVL.IOVD.X_I_In_Elec_Heat.na AND NOT GVL.IOVD.X_I_In_Elec_Heat.e AND NOT GVL.IOVD.X_I_In_Elec_Heat.RangeExcd;
GVL.IOVD.X_I_In_Elec_Heat.x					:= GVL.IICH.X_I_Elec_Heat.x;
GVL.IOVD.X_I_In_Elec_Heat.e					:= GVL.IICH.X_I_Elec_Heat.e;
GVL.IOVD.X_I_In_Elec_Heat.na				:= GVL.IICH.X_I_Elec_Heat.na;
GVL.IOVD.X_I_In_Elec_Heat.RangeExcd			:=  (3212.75 < GVL.IOVD.X_I_In_Elec_Heat.x )OR (0 > GVL.IOVD.X_I_In_Elec_Heat.x);
{endregion}
//-----------------------------------------------------------------------------------------------------------------------------
//-----------------------------------------------------------------------------------------------------------------------------
//MESSAGE------
{region " User Area : Klima_Kontaktor_Kontrol- ID:414"}

//-------SIGNAL -> C_Defrs_Plus_Ct Max: 1 Min: 0 Def: 0 Resolution: 1 Offset: 0
GVL.IOVD.C_Defrs_Plus_Ct.v					:= GVL.SY.S_ECU_Rdy;
GVL.IOVD.C_Defrs_Plus_Ct.x					:= GVL.IOPT.C_Aux_DC_HV_Ct_2_On.x;
//-------SIGNAL -> C_Defrs_Minus_Ct Max: 1 Min: 0 Def: 0 Resolution: 1 Offset: 0
GVL.IOVD.C_Defrs_Minus_Ct.v					:= GVL.SY.S_ECU_Rdy;
GVL.IOVD.C_Defrs_Minus_Ct.x					:= GVL.IOPT.C_Aux_DC_HV_Ct_2_On.x;
//-------SIGNAL -> C_Prheat_Plus_Ct Max: 1 Min: 0 Def: 0 Resolution: 1 Offset: 0
GVL.IOVD.C_Prheat_Plus_Ct.v					:= GVL.SY.S_ECU_Rdy;
GVL.IOVD.C_Prheat_Plus_Ct.x					:= GVL.IOPT.C_Aux_DC_HV_Ct_1_On.x;
//-------SIGNAL -> C_Prheat_Minus_Ct Max: 1 Min: 0 Def: 0 Resolution: 1 Offset: 0
GVL.IOVD.C_Prheat_Minus_Ct.v				:= GVL.SY.S_ECU_Rdy;
GVL.IOVD.C_Prheat_Minus_Ct.x				:= GVL.IOPT.C_Aux_DC_HV_Ct_1_On.x;
//-------SIGNAL -> C_HVAC_Plus_Ct Max: 1 Min: 0 Def: 0 Resolution: 1 Offset: 0
GVL.IOVD.C_HVAC_Plus_Ct.v					:= GVL.SY.S_ECU_Rdy;
GVL.IOVD.C_HVAC_Plus_Ct.x					:= GVL.IOPT.C_Aux_DC_HV_Ct_1_On.x;
//-------SIGNAL -> C_HVAC_Minus_Ct Max: 1 Min: 0 Def: 0 Resolution: 1 Offset: 0
GVL.IOVD.C_HVAC_Minus_Ct.v					:= GVL.SY.S_ECU_Rdy;
GVL.IOVD.C_HVAC_Minus_Ct.x					:= GVL.IOPT.C_Aux_DC_HV_Ct_1_On.x;
//-------SIGNAL -> S_Defrs_Plus_Ct_Deactv Max: 1 Min: 0 Def: 0 Resolution: 1 Offset: 0
GVL.IOVD.S_Defrs_Plus_Ct_Deactv.v			:= GVL.SY.S_ECU_Rdy;
GVL.IOVD.S_Defrs_Plus_Ct_Deactv.x			:= GVL.IIPT.S_Aux_DC_HV_Ct_2_On.x;
//-------SIGNAL -> S_Defrs_Minus_Ct_Deactv Max: 1 Min: 0 Def: 0 Resolution: 1 Offset: 0
GVL.IOVD.S_Defrs_Minus_Ct_Deactv.v			:= GVL.SY.S_ECU_Rdy;
GVL.IOVD.S_Defrs_Minus_Ct_Deactv.x			:= GVL.IIPT.S_Aux_DC_HV_Ct_2_On.x;
//-------SIGNAL -> S_Prheat_Plus_Ct_Deactv Max: 1 Min: 0 Def: 0 Resolution: 1 Offset: 0
GVL.IOVD.S_Prheat_Plus_Ct_Deactv.v			:= GVL.SY.S_ECU_Rdy;
GVL.IOVD.S_Prheat_Plus_Ct_Deactv.x			:= GVL.IIPT.S_Aux_DC_HV_Ct_1_On.x;
//-------SIGNAL -> S_Prheat_Minus_Ct_Deactv Max: 1 Min: 0 Def: 0 Resolution: 1 Offset: 0
GVL.IOVD.S_Prheat_Minus_Ct_Deactv.v			:= GVL.SY.S_ECU_Rdy;
GVL.IOVD.S_Prheat_Minus_Ct_Deactv.x			:= GVL.IIPT.S_Aux_DC_HV_Ct_1_On.x;
//-------SIGNAL -> S_HVAC_Plus_Ct_Deactv Max: 1 Min: 0 Def: 0 Resolution: 1 Offset: 0
GVL.IOVD.S_HVAC_Plus_Ct_Deactv.v			:= GVL.SY.S_ECU_Rdy;
GVL.IOVD.S_HVAC_Plus_Ct_Deactv.x			:= GVL.IIPT.S_Aux_DC_HV_Ct_1_On.x;
//-------SIGNAL -> S_HVAC_Minus_Ct_Deactv Max: 1 Min: 0 Def: 0 Resolution: 1 Offset: 0
GVL.IOVD.S_HVAC_Minus_Ct_Deactv.v			:= GVL.SY.S_ECU_Rdy;
GVL.IOVD.S_HVAC_Minus_Ct_Deactv.x			:= GVL.IIPT.S_Aux_DC_HV_Ct_1_On.x;
//-------SIGNAL -> Z_Btms_Stat Max: 255 Min: 0 Def: 0 Resolution: 1 Offset: 0
GVL.IOVD.Z_Btms_Stat.v						:= GVL.SY.S_ECU_Rdy AND NOT GVL.IOVD.Z_Btms_Stat.e	AND NOT GVL.IOVD.Z_Btms_Stat.na AND NOT GVL.IOVD.Z_Btms_Stat.RangeExcd;
GVL.IOVD.Z_Btms_Stat.e						:= FALSE;
GVL.IOVD.Z_Btms_Stat.na						:= FALSE;
GVL.IOVD.Z_Btms_Stat.RangeExcd				:=  (255 < GVL.IOVD.Z_Btms_Stat.x )OR (0 > GVL.IOVD.Z_Btms_Stat.x);	 
_FB_PACK_8BITS_TO_BYTE_0 (		S_BIT_0 	:= GVL.IICH.Z_BTMS.v AND GVL.IICH.Z_BTMS.x <> 0,
								S_BIT_1		:= GVL.IICH.Z_BTMS.v AND (GVL.IICH.Z_BTMS.x = 1 OR GVL.IICH.Z_BTMS.x = 3),
								S_BIT_2 	:= GVL.IICH.Z_BTMS.v AND GVL.IICH.Z_BTMS.x = 2,
								S_BIT_3 	:= 0,	//Fault
								S_BIT_4 	:= 0, 
								S_BIT_5 	:= 0,
								S_BIT_6 	:= 0,
								S_BIT_7 	:= 0,
								X_BYTE_0 	=> GVL.IOVD.Z_Btms_Stat.x);								 
//-------SIGNAL -> Z_HvacDrv_Stat Max: 255 Min: 0 Def: 0 Resolution: 1 Offset: 0
GVL.IOVD.Z_HvacDrv_Stat.v					:= GVL.SY.S_ECU_Rdy AND NOT GVL.IOVD.Z_HvacDrv_Stat.e	AND NOT GVL.IOVD.Z_HvacDrv_Stat.na AND NOT GVL.IOVD.Z_HvacDrv_Stat.RangeExcd;
GVL.IOVD.Z_HvacDrv_Stat.e					:= FALSE;
GVL.IOVD.Z_HvacDrv_Stat.na					:= FALSE;
GVL.IOVD.Z_HvacDrv_Stat.RangeExcd			:=  (255 < GVL.IOVD.Z_HvacDrv_Stat.x )OR (0 > GVL.IOVD.Z_HvacDrv_Stat.x);	 
_FB_PACK_8BITS_TO_BYTE_1 (		S_BIT_0 	:= GVL.IICH.Z_Act_Op_Mode.x = 14,	//Force mode
								S_BIT_1		:= GVL.IICH.S_Drv_Cool.x OR GVL.IICH.S_Drv_Heat.x OR GVL.IICH.S_Drv_Ven.x,	//On
								S_BIT_2 	:= GVL.IICH.S_Mn_Swc_Actv.x,		//Supply OK
								S_BIT_3 	:= GVL.IICH.S_Drv_Cool.x,			//Cooling
								S_BIT_4 	:= GVL.IICH.S_Drv_Heat.x, 			//Heating
								S_BIT_5 	:= GVL.IICH.S_Drv_Ven.x,			//Ventilation
								S_BIT_6 	:= 0,								//ECO mode
								S_BIT_7 	:= GVL.IICH.N_Actv_Err.x <> 0,		//Error
								X_BYTE_0 	=> GVL.IOVD.Z_HvacDrv_Stat.x);						  										 																									 
//-------SIGNAL -> Z_HvacPass1_Stat Max: 255 Min: 0 Def: 0 Resolution: 1 Offset: 0
GVL.IOVD.Z_HvacPass1_Stat.v					:= GVL.SY.S_ECU_Rdy AND NOT GVL.IOVD.Z_HvacPass1_Stat.e	AND NOT GVL.IOVD.Z_HvacPass1_Stat.na AND NOT GVL.IOVD.Z_HvacPass1_Stat.RangeExcd;
GVL.IOVD.Z_HvacPass1_Stat.e					:= FALSE;
GVL.IOVD.Z_HvacPass1_Stat.na				:= FALSE;
GVL.IOVD.Z_HvacPass1_Stat.RangeExcd			:=  (255 < GVL.IOVD.Z_HvacPass1_Stat.x )OR (0 > GVL.IOVD.Z_HvacPass1_Stat.x);	 
_FB_PACK_8BITS_TO_BYTE_2 (		S_BIT_0 	:= GVL.IICH.Z_Act_Op_Mode.v AND GVL.IICH.Z_Act_Op_Mode.x = 14,	//Force mode
								S_BIT_1		:= GVL.IICH.Z_Act_Op_Mode.v AND GVL.IICH.Z_Act_Op_Mode.x <> 15,	//On
								S_BIT_2 	:= GVL.IICH.S_Mn_Swc_Actv.x,		//Supply OK
								S_BIT_3 	:= GVL.IICH.Z_Act_Op_Mode.v AND GVL.IICH.Z_Act_Op_Mode.x = 2,	//Cooling
								S_BIT_4 	:= GVL.IICH.Z_Act_Op_Mode.v AND GVL.IICH.Z_Act_Op_Mode.x = 1, 	//Heating
								S_BIT_5 	:= GVL.IICH.Z_Act_Op_Mode.v AND GVL.IICH.Z_Act_Op_Mode.x = 0,	//Ventilation
								S_BIT_6 	:= GVL.IICH.Z_Act_Op_Mode.v AND GVL.IICH.Z_Act_Op_Mode.x = 5,	//Auto mode
								S_BIT_7 	:= GVL.IICH.N_Actv_Err.x <> 0,		//Error
								X_BYTE_0 	=> GVL.IOVD.Z_HvacPass1_Stat.x);
//-------SIGNAL -> Z_HvacPass2_Stat Max: 255 Min: 0 Def: 0 Resolution: 1 Offset: 0
GVL.IOVD.Z_HvacPass2_Stat.v					:= GVL.SY.S_ECU_Rdy AND NOT GVL.IOVD.Z_HvacPass2_Stat.e	AND NOT GVL.IOVD.Z_HvacPass2_Stat.na AND NOT GVL.IOVD.Z_HvacPass2_Stat.RangeExcd;
GVL.IOVD.Z_HvacPass2_Stat.x					:= 0;
GVL.IOVD.Z_HvacPass2_Stat.e					:= FALSE;
GVL.IOVD.Z_HvacPass2_Stat.na				:= FALSE;
GVL.IOVD.Z_HvacPass2_Stat.RangeExcd			:=  (255 < GVL.IOVD.Z_HvacPass2_Stat.x )OR (0 > GVL.IOVD.Z_HvacPass2_Stat.x);	 
//-------SIGNAL -> Z_Elec_Heaters_Stat Max: 255 Min: 0 Def: 0 Resolution: 1 Offset: 0
GVL.IOVD.Z_Elec_Heaters_Stat.v				:= GVL.SY.S_ECU_Rdy AND NOT GVL.IOVD.Z_Elec_Heaters_Stat.e	AND NOT GVL.IOVD.Z_Elec_Heaters_Stat.na AND NOT GVL.IOVD.Z_Elec_Heaters_Stat.RangeExcd;
GVL.IOVD.Z_Elec_Heaters_Stat.e				:= FALSE;
GVL.IOVD.Z_Elec_Heaters_Stat.na				:= FALSE;
GVL.IOVD.Z_Elec_Heaters_Stat.RangeExcd		:=  (255 < GVL.IOVD.Z_Elec_Heaters_Stat.x )OR (0 > GVL.IOVD.Z_Elec_Heaters_Stat.x);	 
_FB_PACK_8BITS_TO_BYTE_3 (		S_BIT_0 	:= GVL.IICH.C_Elec_Heat_1_On.x,							//Electric heater 1 on
								S_BIT_1		:= GVL.IICH.S_Elec_Heat_HV_Loop_Actv.v AND (NOT GVL.IICH.S_Elec_Heat_HV_Loop_Actv.x OR NOT GVL.IICH.S_Elec_Heat_Sfty_Cnt_Actv.x),	//Electric heater 1 fault
								S_BIT_2 	:= GVL.IICH.C_Elec_Heat_2_On.x,							//Electric heater 2 on
								S_BIT_3 	:= GVL.IICH.S_Elec_Heat_HV_Loop_Actv.v AND (NOT GVL.IICH.S_Elec_Heat_HV_Loop_Actv.x OR NOT GVL.IICH.S_Elec_Heat_Sfty_Cnt_Actv.x),	//Electric heater 2 fault
								S_BIT_4 	:= 0,	//Electric heater 3 on
								S_BIT_5 	:= 0,	//Electric heater 3 fault
								S_BIT_6 	:= 0,	//Timer active
								S_BIT_7 	:= 0,	//Spare
								X_BYTE_0 	=> GVL.IOVD.Z_Elec_Heaters_Stat.x);
//-------SIGNAL -> Z_Flr_Heaters_Stat_1 Max: 255 Min: 0 Def: 0 Resolution: 1 Offset: 0
GVL.IOVD.Z_Flr_Heaters_Stat_1.v				:= GVL.SY.S_ECU_Rdy AND NOT GVL.IOVD.Z_Flr_Heaters_Stat_1.e	AND NOT GVL.IOVD.Z_Flr_Heaters_Stat_1.na AND NOT GVL.IOVD.Z_Flr_Heaters_Stat_1.RangeExcd;
GVL.IOVD.Z_Flr_Heaters_Stat_1.e				:= FALSE;
GVL.IOVD.Z_Flr_Heaters_Stat_1.na			:= FALSE;
GVL.IOVD.Z_Flr_Heaters_Stat_1.RangeExcd		:=  (255 < GVL.IOVD.Z_Flr_Heaters_Stat_1.x )OR (0 > GVL.IOVD.Z_Flr_Heaters_Stat_1.x);
_FB_PACK_8BITS_TO_BYTE_4 (		S_BIT_0 	:= GVL.IIVD.S_Flr_Heat_1.x,													// Floor heater 1 active
								S_BIT_1		:= GVL.IIVD.S_ER_Flr_Heat_1_Thstat.x OR GVL.IIVD.S_Flr_Heat_1_Fus_Blw.x,	// Floor heater 1 fault
								S_BIT_2 	:= GVL.IIVD.S_Flr_Heat_2.x,													// Floor heater 2 active
								S_BIT_3 	:= GVL.IIVD.S_ER_Flr_Heat_2_Thstat.x OR GVL.IIVD.S_Flr_Heat_2_Fus_Blw.x,	// Floor heater 2 fault
								S_BIT_4 	:= GVL.IIVD.S_Flr_Heat_3.x,													// Floor heater 3 active
								S_BIT_5 	:= GVL.IIVD.S_ER_Flr_Heat_3_Thstat.x OR GVL.IIVD.S_Flr_Heat_3_Fus_Blw.x,	// Floor heater 3 fault
								S_BIT_6 	:= GVL.IIVD.S_Flr_Heat_4.x,													// Floor heater 4 active
								S_BIT_7 	:= GVL.IIVD.S_ER_Flr_Heat_4_Thstat.x OR GVL.IIVD.S_Flr_Heat_4_Fus_Blw.x,	// Floor heater 4 fault
								X_BYTE_0 	=> GVL.IOVD.Z_Flr_Heaters_Stat_1.x);								 
//-------SIGNAL -> Z_Flr_Heaters_Stat_2 Max: 255 Min: 0 Def: 0 Resolution: 1 Offset: 0
GVL.IOVD.Z_Flr_Heaters_Stat_2.v				:= GVL.SY.S_ECU_Rdy AND NOT GVL.IOVD.Z_Flr_Heaters_Stat_2.e	AND NOT GVL.IOVD.Z_Flr_Heaters_Stat_2.na AND NOT GVL.IOVD.Z_Flr_Heaters_Stat_2.RangeExcd;
GVL.IOVD.Z_Flr_Heaters_Stat_2.x				:= 0;
GVL.IOVD.Z_Flr_Heaters_Stat_2.e				:= FALSE;
GVL.IOVD.Z_Flr_Heaters_Stat_2.na			:= FALSE;
GVL.IOVD.Z_Flr_Heaters_Stat_2.RangeExcd		:= (255 < GVL.IOVD.Z_Flr_Heaters_Stat_1.x )OR (0 > GVL.IOVD.Z_Flr_Heaters_Stat_1.x);	
{endregion}
//-----------------------------------------------------------------------------------------------------------------------------
//-----------------------------------------------------------------------------------------------------------------------------
//MESSAGE------
{region " User Area : HVAC_Parameters_1- ID:415"}
//-------SIGNAL -> P_X_T_Max_Bat_BTMS_Heat Max: 250 Min: 0 Def: 0 Resolution: 1 Offset: 0
GVL.IOVD.P_X_T_Max_Bat_BTMS_Heat.v				:= GVL.SY.S_ECU_Rdy AND NOT GVL.IOVD.P_X_T_Max_Bat_BTMS_Heat.na AND NOT GVL.IOVD.P_X_T_Max_Bat_BTMS_Heat.e AND NOT GVL.IOVD.P_X_T_Max_Bat_BTMS_Heat.RangeExcd;
GVL.IOVD.P_X_T_Max_Bat_BTMS_Heat.x				:= GVL.EG.P_X_T_Max_Bat_BTMS_Heat;
GVL.IOVD.P_X_T_Max_Bat_BTMS_Heat.e				:= FALSE;
GVL.IOVD.P_X_T_Max_Bat_BTMS_Heat.na				:= GVL.IIVD.S_TmOut_Parametre_1_0X263;
GVL.IOVD.P_X_T_Max_Bat_BTMS_Heat.RangeExcd		:= (250 < GVL.IOVD.P_X_T_Max_Bat_BTMS_Heat.x) OR (0 > GVL.IOVD.P_X_T_Max_Bat_BTMS_Heat.x);

//-------SIGNAL -> P_X_T_Max_Bat_BTMS_Cool Max: 250 Min: 0 Def: 0 Resolution: 1 Offset: 0
GVL.IOVD.P_X_T_Max_Bat_BTMS_Cool.v				:= GVL.SY.S_ECU_Rdy AND NOT GVL.IOVD.P_X_T_Max_Bat_BTMS_Cool.na AND NOT GVL.IOVD.P_X_T_Max_Bat_BTMS_Cool.e AND NOT GVL.IOVD.P_X_T_Max_Bat_BTMS_Cool.RangeExcd;
GVL.IOVD.P_X_T_Max_Bat_BTMS_Cool.x				:= GVL.EG.P_X_T_Max_Bat_BTMS_Cool;
GVL.IOVD.P_X_T_Max_Bat_BTMS_Cool.e				:= FALSE;
GVL.IOVD.P_X_T_Max_Bat_BTMS_Cool.na				:= GVL.IIVD.S_TmOut_Parametre_1_0X263;
GVL.IOVD.P_X_T_Max_Bat_BTMS_Cool.RangeExcd		:= (250 < GVL.IOVD.P_X_T_Max_Bat_BTMS_Cool.x) OR (0 > GVL.IOVD.P_X_T_Max_Bat_BTMS_Cool.x);

//-------SIGNAL -> P_X_T_Max_Wtr_BTMS_Heat Max: 250 Min: 0 Def: 0 Resolution: 1 Offset: 0
GVL.IOVD.P_X_T_Max_Wtr_BTMS_Heat.v				:= GVL.SY.S_ECU_Rdy AND NOT GVL.IOVD.P_X_T_Max_Wtr_BTMS_Heat.na AND NOT GVL.IOVD.P_X_T_Max_Wtr_BTMS_Heat.e AND NOT GVL.IOVD.P_X_T_Max_Wtr_BTMS_Heat.RangeExcd;
GVL.IOVD.P_X_T_Max_Wtr_BTMS_Heat.x				:= GVL.EG.P_X_T_Max_Wtr_BTMS_Heat;
GVL.IOVD.P_X_T_Max_Wtr_BTMS_Heat.e				:= FALSE;
GVL.IOVD.P_X_T_Max_Wtr_BTMS_Heat.na				:= GVL.IIVD.S_TmOut_Parametre_1_0X263;
GVL.IOVD.P_X_T_Max_Wtr_BTMS_Heat.RangeExcd		:= (250 < GVL.IOVD.P_X_T_Max_Wtr_BTMS_Heat.x) OR (0 > GVL.IOVD.P_X_T_Max_Wtr_BTMS_Heat.x);

//-------SIGNAL -> P_X_T_Max_Wtr_BTMS_Cool Max: 250 Min: 0 Def: 0 Resolution: 1 Offset: 0
GVL.IOVD.P_X_T_Max_Wtr_BTMS_Cool.v				:= GVL.SY.S_ECU_Rdy AND NOT GVL.IOVD.P_X_T_Max_Wtr_BTMS_Cool.na AND NOT GVL.IOVD.P_X_T_Max_Wtr_BTMS_Cool.e AND NOT GVL.IOVD.P_X_T_Max_Wtr_BTMS_Cool.RangeExcd;
GVL.IOVD.P_X_T_Max_Wtr_BTMS_Cool.x				:= GVL.EG.P_X_T_Max_Wtr_BTMS_Cool;
GVL.IOVD.P_X_T_Max_Wtr_BTMS_Cool.e				:= FALSE;
GVL.IOVD.P_X_T_Max_Wtr_BTMS_Cool.na				:= GVL.IIVD.S_TmOut_Parametre_1_0X263;
GVL.IOVD.P_X_T_Max_Wtr_BTMS_Cool.RangeExcd		:= (250 < GVL.IOVD.P_X_T_Max_Wtr_BTMS_Cool.x) OR (0 > GVL.IOVD.P_X_T_Max_Wtr_BTMS_Cool.x);

//-------SIGNAL -> P_X_T_Flr_Heat_Lim Max: 250 Min: 0 Def: 0 Resolution: 1 Offset: 0
GVL.IOVD.P_X_T_Flr_Heat_Lim.v					:= GVL.SY.S_ECU_Rdy AND NOT GVL.IOVD.P_X_T_Flr_Heat_Lim.na AND NOT GVL.IOVD.P_X_T_Flr_Heat_Lim.e AND NOT GVL.IOVD.P_X_T_Flr_Heat_Lim.RangeExcd;
GVL.IOVD.P_X_T_Flr_Heat_Lim.x					:= GVL.EG.P_X_T_Flr_Heat_Lim;
GVL.IOVD.P_X_T_Flr_Heat_Lim.e					:= FALSE;
GVL.IOVD.P_X_T_Flr_Heat_Lim.na					:= GVL.IIVD.S_TmOut_Parametre_1_0X263;
GVL.IOVD.P_X_T_Flr_Heat_Lim.RangeExcd			:= (250 < GVL.IOVD.P_X_T_Flr_Heat_Lim.x) OR (0 > GVL.IOVD.P_X_T_Flr_Heat_Lim.x);
{endregion}
//-----------------------------------------------------------------------------------------------------------------------------
//-----------------------------------------------------------------------------------------------------------------------------
//MESSAGE------
{region " User Area : HVAC_Water_Temperature- ID:416"}

//-------SIGNAL -> X_T_BTMS_Wtr_Snsr_1 Max: 150 Min: -40 Def: 0 Resolution: 1 Offset: -40
GVL.IOVD.X_T_BTMS_Wtr_Snsr_1.v					:= GVL.SY.S_ECU_Rdy AND NOT GVL.IOVD.X_T_BTMS_Wtr_Snsr_1.e AND NOT GVL.IOVD.X_T_BTMS_Wtr_Snsr_1.na AND NOT GVL.IOVD.X_T_BTMS_Wtr_Snsr_1.RangeExcd;
GVL.IOVD.X_T_BTMS_Wtr_Snsr_1.x					:= UDINT_TO_REAL(DWORD_TO_UDINT(GVL.IIRE.X_T_BTMS_Wtr_Snsr_In_Sd_Frnt_Md.value));
GVL.IOVD.X_T_BTMS_Wtr_Snsr_1.e					:= GVL.IIRE.X_T_BTMS_Wtr_Snsr_In_Sd_Frnt_Md.error <> lib500_types.IO_ERRORTYPE.IO_E_OK;
GVL.IOVD.X_T_BTMS_Wtr_Snsr_1.na					:= FALSE;
GVL.IOVD.X_T_BTMS_Wtr_Snsr_1.RangeExcd			:= (150 < GVL.IOVD.X_T_BTMS_Wtr_Snsr_1.x) OR (-40 > GVL.IOVD.X_T_BTMS_Wtr_Snsr_1.x);

//-------SIGNAL -> X_T_BTMS_Wtr_Snsr_2 Max: 150 Min: -40 Def: 0 Resolution: 1 Offset: -40
GVL.IOVD.X_T_BTMS_Wtr_Snsr_2.v					:= GVL.SY.S_ECU_Rdy AND NOT GVL.IOVD.X_T_BTMS_Wtr_Snsr_2.e AND NOT GVL.IOVD.X_T_BTMS_Wtr_Snsr_2.na AND NOT GVL.IOVD.X_T_BTMS_Wtr_Snsr_2.RangeExcd;
GVL.IOVD.X_T_BTMS_Wtr_Snsr_2.x					:= UDINT_TO_REAL(DWORD_TO_UDINT(GVL.IIRE.X_T_BTMS_Wtr_Snsr_In_Sd.value));
GVL.IOVD.X_T_BTMS_Wtr_Snsr_2.e					:= GVL.IIRE.X_T_BTMS_Wtr_Snsr_In_Sd.error <> lib500_types.IO_ERRORTYPE.IO_E_OK;
GVL.IOVD.X_T_BTMS_Wtr_Snsr_2.na					:= FALSE;
GVL.IOVD.X_T_BTMS_Wtr_Snsr_2.RangeExcd			:= (150 < GVL.IOVD.X_T_BTMS_Wtr_Snsr_2.x) OR (-40 > GVL.IOVD.X_T_BTMS_Wtr_Snsr_2.x);
{endregion}
//-----------------------------------------------------------------------------------------------------------------------------
//-----------------------------------------------------------------------------------------------------------------------------
//MESSAGE------
{region " User Area : Arac_Menzil- ID:4C0"}

//-------SIGNAL -> X_Distn_Bat_Drvn Max: 65000 Min: 0 Def: 0 Resolution: 1 Offset: 0
GVL.IOVD.X_Distn_Bat_Drvn.v					:= GVL.SY.S_ECU_Rdy AND NOT GVL.IOVD.X_Distn_Bat_Drvn.e	AND NOT GVL.IOVD.X_Distn_Bat_Drvn.na AND NOT GVL.IOVD.X_Distn_Bat_Drvn.RangeExcd;
GVL.IOVD.X_Distn_Bat_Drvn.x					:= GVL.PV.X_Dist_Bat;
GVL.IOVD.X_Distn_Bat_Drvn.e					:= FALSE;
GVL.IOVD.X_Distn_Bat_Drvn.na				:= FALSE;
GVL.IOVD.X_Distn_Bat_Drvn.RangeExcd			:= (65000 < GVL.IOVD.X_Distn_Bat_Drvn.x) OR (0 > GVL.IOVD.X_Distn_Bat_Drvn.x);
//-------SIGNAL -> X_Distn_Rmn Max: 65000 Min: 0 Def: 0 Resolution: 1 Offset: 0
GVL.IOVD.X_Distn_Rmn.v						:= GVL.SY.S_ECU_Rdy AND NOT GVL.IOVD.X_Distn_Rmn.e	AND NOT GVL.IOVD.X_Distn_Rmn.na AND NOT GVL.IOVD.X_Distn_Rmn.RangeExcd;
GVL.IOVD.X_Distn_Rmn.x						:= GVL.PV.X_Dist_Rmn;
GVL.IOVD.X_Distn_Rmn.e						:= FALSE;
GVL.IOVD.X_Distn_Rmn.na						:= FALSE;
GVL.IOVD.X_Distn_Rmn.RangeExcd				:= (65000 < GVL.IOVD.X_Distn_Rmn.x) OR (0 > GVL.IOVD.X_Distn_Rmn.x);
//-------SIGNAL -> X_Distn_Cat_Drvn Max: 4.21108e+09 Min: 0 Def: 0 Resolution: 1 Offset: 0
GVL.IOVD.X_Distn_Cat_Drvn.v					:= GVL.SY.S_ECU_Rdy AND NOT GVL.IOVD.X_Distn_Cat_Drvn.e	AND NOT GVL.IOVD.X_Distn_Cat_Drvn.na AND NOT GVL.IOVD.X_Distn_Cat_Drvn.RangeExcd;
GVL.IOVD.X_Distn_Cat_Drvn.x					:= GVL.PV.X_Dist_Cat;
GVL.IOVD.X_Distn_Cat_Drvn.e					:= FALSE;
GVL.IOVD.X_Distn_Cat_Drvn.na				:= FALSE;
GVL.IOVD.X_Distn_Cat_Drvn.RangeExcd			:= (4211081215 < GVL.IOVD.X_Distn_Cat_Drvn.x) OR (0 > GVL.IOVD.X_Distn_Cat_Drvn.x);
{endregion}
//-----------------------------------------------------------------------------------------------------------------------------
//-----------------------------------------------------------------------------------------------------------------------------
//MESSAGE------
{region " User Area : Arac_Odometre- ID:4C1"}

//-------SIGNAL -> X_Om Max: 4.21108e+08 Min: 0 Def: 0 Resolution: 1 Offset: 0
GVL.IOVD.X_Om.v								:= GVL.SY.S_ECU_Rdy AND NOT GVL.IOVD.X_Om.e	AND NOT GVL.IOVD.X_Om.na AND NOT GVL.IOVD.X_Om.RangeExcd;
GVL.IOVD.X_Om.x								:= GVL.PV.X_Odo;
GVL.IOVD.X_Om.e								:= FALSE;
GVL.IOVD.X_Om.na							:= FALSE;
GVL.IOVD.X_Om.RangeExcd						:= (421108121.5 < GVL.IOVD.X_Om.x) OR (0 > GVL.IOVD.X_Om.x);
{endregion}
//-----------------------------------------------------------------------------------------------------------------------------
//-----------------------------------------------------------------------------------------------------------------------------
//MESSAGE------
{region " User Area : Arac_Surus_Enerji- ID:4C3"}

//-------SIGNAL -> X_E_Tr Max: 4.21108e+08 Min: 0 Def: 0 Resolution: 0.1 Offset: 0
GVL.IOVD.X_E_Tr.v							:= GVL.SY.S_ECU_Rdy AND NOT GVL.IOVD.X_E_Tr.e	AND NOT GVL.IOVD.X_E_Tr.na AND NOT GVL.IOVD.X_E_Tr.RangeExcd;
GVL.IOVD.X_E_Tr.x							:= GVL.PV.X_E_Tr;
GVL.IOVD.X_E_Tr.e							:= FALSE;
GVL.IOVD.X_E_Tr.na							:= FALSE;
GVL.IOVD.X_E_Tr.RangeExcd					:= (421108121.5 < GVL.IOVD.X_E_Tr.x) OR (0 > GVL.IOVD.X_E_Tr.x);
//-------SIGNAL -> X_E_Regn Max: 4.21108e+08 Min: 0 Def: 0 Resolution: 0.1 Offset: 0
GVL.IOVD.X_E_Regn.v							:= GVL.SY.S_ECU_Rdy AND NOT GVL.IOVD.X_E_Regn.e	AND NOT GVL.IOVD.X_E_Regn.na AND NOT GVL.IOVD.X_E_Regn.RangeExcd;
GVL.IOVD.X_E_Regn.x							:= GVL.PV.X_E_Regn;
GVL.IOVD.X_E_Regn.e							:= FALSE;
GVL.IOVD.X_E_Regn.na						:= FALSE;
GVL.IOVD.X_E_Regn.RangeExcd					:= (421108121.5 < GVL.IOVD.X_E_Regn.x) OR (0 > GVL.IOVD.X_E_Regn.x);
{endregion}
//-----------------------------------------------------------------------------------------------------------------------------
//-----------------------------------------------------------------------------------------------------------------------------
//MESSAGE------
{region " User Area : Arac_Tuketilen_Enerji_1- ID:4C4"}

//-------SIGNAL -> X_E_Aux_DC Max: 4.21108e+08 Min: 0 Def: 0 Resolution: 0.1 Offset: 0
GVL.IOVD.X_E_Aux_DC.v						:= GVL.SY.S_ECU_Rdy AND NOT GVL.IOVD.X_E_Aux_DC.e	AND NOT GVL.IOVD.X_E_Aux_DC.na AND NOT GVL.IOVD.X_E_Aux_DC.RangeExcd;
GVL.IOVD.X_E_Aux_DC.x						:= GVL.PV.X_E_Aux_DC;
GVL.IOVD.X_E_Aux_DC.e						:= FALSE;
GVL.IOVD.X_E_Aux_DC.na						:= FALSE;
GVL.IOVD.X_E_Aux_DC.RangeExcd				:= (421108121.5 < GVL.IOVD.X_E_Aux_DC.x) OR (0 > GVL.IOVD.X_E_Aux_DC.x);
//-------SIGNAL -> X_E_Aux_DC_24V Max: 4.21108e+08 Min: 0 Def: 0 Resolution: 0.1 Offset: 0
GVL.IOVD.X_E_Aux_DC_24V.v					:= GVL.SY.S_ECU_Rdy AND NOT GVL.IOVD.X_E_Aux_DC_24V.e	AND NOT GVL.IOVD.X_E_Aux_DC_24V.na AND NOT GVL.IOVD.X_E_Aux_DC_24V.RangeExcd;
GVL.IOVD.X_E_Aux_DC_24V.x					:= GVL.PV.X_E_Aux_DC_24V;
GVL.IOVD.X_E_Aux_DC_24V.e					:= FALSE;
GVL.IOVD.X_E_Aux_DC_24V.na					:= FALSE;
GVL.IOVD.X_E_Aux_DC_24V.RangeExcd			:= (421108121.5 < GVL.IOVD.X_E_Aux_DC_24V.x) OR (0 > GVL.IOVD.X_E_Aux_DC_24V.x);
{endregion}
//-----------------------------------------------------------------------------------------------------------------------------
//-----------------------------------------------------------------------------------------------------------------------------
//MESSAGE------
{region " User Area : Arac_Tuketilen_Enerji_2- ID:4C5"}

//-------SIGNAL -> X_E_Aux_AC Max: 4.21108e+08 Min: 0 Def: 0 Resolution: 0.1 Offset: 0
GVL.IOVD.X_E_Aux_AC.v						:= GVL.SY.S_ECU_Rdy AND NOT GVL.IOVD.X_E_Aux_AC.e	AND NOT GVL.IOVD.X_E_Aux_AC.na AND NOT GVL.IOVD.X_E_Aux_AC.RangeExcd;
GVL.IOVD.X_E_Aux_AC.x						:= GVL.PV.X_E_Aux_AC;
GVL.IOVD.X_E_Aux_AC.e						:= FALSE;
GVL.IOVD.X_E_Aux_AC.na						:= FALSE;
GVL.IOVD.X_E_Aux_AC.RangeExcd				:= (421108121.5 < GVL.IOVD.X_E_Aux_AC.x) OR (0 > GVL.IOVD.X_E_Aux_AC.x);
//-------SIGNAL -> X_E_Cosu Max: 4.21108e+08 Min: 0 Def: 0 Resolution: 0.1 Offset: 0
GVL.IOVD.X_E_Cosu.v							:= GVL.SY.S_ECU_Rdy AND NOT GVL.IOVD.X_E_Cosu.e	AND NOT GVL.IOVD.X_E_Cosu.na AND NOT GVL.IOVD.X_E_Cosu.RangeExcd;
GVL.IOVD.X_E_Cosu.x							:= GVL.PV.X_E_Cosu;
GVL.IOVD.X_E_Cosu.e							:= FALSE;
GVL.IOVD.X_E_Cosu.na						:= FALSE;
GVL.IOVD.X_E_Cosu.RangeExcd					:= (421108121.5 < GVL.IOVD.X_E_Cosu.x) OR (0 > GVL.IOVD.X_E_Cosu.x);
{endregion}
//-----------------------------------------------------------------------------------------------------------------------------
//-----------------------------------------------------------------------------------------------------------------------------
//MESSAGE------
{region " User Area : Arac_Kapasite- ID:4C6"}

//-------SIGNAL -> X_Capcty_Act Max: 4.21108e+08 Min: 0 Def: 0 Resolution: 0.1 Offset: 0
GVL.IOVD.X_Capcty_Act.v						:= GVL.SY.S_ECU_Rdy AND NOT GVL.IOVD.X_Capcty_Act.e	AND NOT GVL.IOVD.X_Capcty_Act.na AND NOT GVL.IOVD.X_Capcty_Act.RangeExcd;
GVL.IOVD.X_Capcty_Act.x						:= GVL.PV.X_E_Act;
GVL.IOVD.X_Capcty_Act.e						:= FALSE;
GVL.IOVD.X_Capcty_Act.na					:= FALSE;
GVL.IOVD.X_Capcty_Act.RangeExcd				:= (421108121.5 < GVL.IOVD.X_Capcty_Act.x) OR (0 > GVL.IOVD.X_Capcty_Act.x);
//-------SIGNAL -> X_Capcty_Rmn Max: 4.21108e+08 Min: 0 Def: 0 Resolution: 0.1 Offset: 0
GVL.IOVD.X_Capcty_Rmn.v						:= GVL.SY.S_ECU_Rdy AND NOT GVL.IOVD.X_Capcty_Rmn.e	AND NOT GVL.IOVD.X_Capcty_Rmn.na AND NOT GVL.IOVD.X_Capcty_Rmn.RangeExcd;
GVL.IOVD.X_Capcty_Rmn.x						:= 0;
GVL.IOVD.X_Capcty_Rmn.e						:= FALSE;
GVL.IOVD.X_Capcty_Rmn.na					:= FALSE;
GVL.IOVD.X_Capcty_Rmn.RangeExcd				:= (421108121.5 < GVL.IOVD.X_Capcty_Rmn.x) OR (0 > GVL.IOVD.X_Capcty_Rmn.x);
{endregion}
//-----------------------------------------------------------------------------------------------------------------------------
//-----------------------------------------------------------------------------------------------------------------------------
//MESSAGE------
{region " User Area : Arac_Sureler- ID:4C7"}

//-------SIGNAL -> X_Tm_Bat_Drvn Max: 65000 Min: 0 Def: 0 Resolution: 1 Offset: 0
GVL.IOVD.X_Tm_Bat_Drvn.v					:= GVL.SY.S_ECU_Rdy AND NOT GVL.IOVD.X_Tm_Bat_Drvn.e	AND NOT GVL.IOVD.X_Tm_Bat_Drvn.na AND NOT GVL.IOVD.X_Tm_Bat_Drvn.RangeExcd;
GVL.IOVD.X_Tm_Bat_Drvn.x					:= GVL.PV.X_Tm_Bat_Drvn;
GVL.IOVD.X_Tm_Bat_Drvn.e					:= FALSE;
GVL.IOVD.X_Tm_Bat_Drvn.na					:= FALSE;
GVL.IOVD.X_Tm_Bat_Drvn.RangeExcd			:= (65000 < GVL.IOVD.X_Tm_Bat_Drvn.x) OR (0 > GVL.IOVD.X_Tm_Bat_Drvn.x);
//-------SIGNAL -> X_Tm_Cat_Drvn Max: 65000 Min: 0 Def: 0 Resolution: 1 Offset: 0
GVL.IOVD.X_Tm_Cat_Drvn.v					:= GVL.SY.S_ECU_Rdy AND NOT GVL.IOVD.X_Tm_Cat_Drvn.e	AND NOT GVL.IOVD.X_Tm_Cat_Drvn.na AND NOT GVL.IOVD.X_Tm_Cat_Drvn.RangeExcd;
GVL.IOVD.X_Tm_Cat_Drvn.x					:= GVL.PV.X_Tm_Cat_Drvn;
GVL.IOVD.X_Tm_Cat_Drvn.e					:= FALSE;
GVL.IOVD.X_Tm_Cat_Drvn.na					:= FALSE;
GVL.IOVD.X_Tm_Cat_Drvn.RangeExcd			:= (65000 < GVL.IOVD.X_Tm_Cat_Drvn.x) OR (0 > GVL.IOVD.X_Tm_Cat_Drvn.x);
//-------SIGNAL -> X_Tm_Wt Max: 65000 Min: 0 Def: 0 Resolution: 1 Offset: 0
GVL.IOVD.X_Tm_Wt.v							:= GVL.SY.S_ECU_Rdy AND NOT GVL.IOVD.X_Tm_Wt.e	AND NOT GVL.IOVD.X_Tm_Wt.na AND NOT GVL.IOVD.X_Tm_Wt.RangeExcd;
GVL.IOVD.X_Tm_Wt.x							:= GVL.PV.X_Tm_Wt;
GVL.IOVD.X_Tm_Wt.e							:= FALSE;
GVL.IOVD.X_Tm_Wt.na							:= FALSE;
GVL.IOVD.X_Tm_Wt.RangeExcd					:= (65000 < GVL.IOVD.X_Tm_Wt.x) OR (0 > GVL.IOVD.X_Tm_Wt.x);
//-------SIGNAL -> X_Tm_HVAC_On Max: 65000 Min: 0 Def: 0 Resolution: 1 Offset: 0
GVL.IOVD.X_Tm_HVAC_On.v						:= GVL.SY.S_ECU_Rdy AND NOT GVL.IOVD.X_Tm_HVAC_On.e	AND NOT GVL.IOVD.X_Tm_HVAC_On.na AND NOT GVL.IOVD.X_Tm_HVAC_On.RangeExcd;
GVL.IOVD.X_Tm_HVAC_On.x						:= DINT_TO_REAL(TRUNC(GVL.PV.X_Tm_Tot_HVAC_On / 60));		// PR1006_REV_002637_TIMTRO
GVL.IOVD.X_Tm_HVAC_On.e						:= FALSE;
GVL.IOVD.X_Tm_HVAC_On.na					:= FALSE;
GVL.IOVD.X_Tm_HVAC_On.RangeExcd				:= (65000 < GVL.IOVD.X_Tm_HVAC_On.x) OR (0 > GVL.IOVD.X_Tm_HVAC_On.x);
{endregion}
//-----------------------------------------------------------------------------------------------------------------------------
//-----------------------------------------------------------------------------------------------------------------------------
//MESSAGE------
{region " User Area : Arac_Toplam_Tuketilen_Enerji- ID:4C8"}

